(* CoDeSys 2.3.9.42 project: dev2.pro *)
(* Author: JvL *)
(* Libraries: ifm_RAWCan\ifm_RAWCan_NT_V020004.lib 7.6.24 16:48:07, ifm_CR0403\ifm_CR0403_V030400.lib 31.5.24 17:04:27, ifm_CANopen\ifm_NetVarLib_NT_V020004.lib 7.6.24 16:46:42, standard.lib 4.10.05 11:14:46, SysLibCallback.lib 7.6.24 16:43:25, 3S_CANOPENNETVAR.LIB 7.6.24 16:46:41, Iecsfc.lib 13.4.06 15:51:28, Util.lib 7.6.24 16:43:26, ifm_CANopen\3S_CANopenManager.lib 7.6.24 16:46:41, ifm_CANopen\3S_CanDrv.lib 7.6.24 16:46:41 *)

(* PLC configuration (modules and I/O channels)
Configuration [LocalConfiguration] node 0, in %IB0 out %QB0 {IFM_PARAM_WORD_TIME = 0}
AT %IB0 [ChInputBool] Input 00 Bit
AT %IB1 [ChInputBool] Input 01 Bit
AT %IB2 [ChInputBool] Input 02 Bit
AT %IB3 [ChInputBool] Input 03 Bit
IGNITION_KEY AT %IB4 [ChInputBool] Input 04 Bit
CHARGER_INPUT AT %IB5 [ChInputBool] Input 05 Bit
BATTERY1_IGNITION AT %IB6 [ChInputBool] Input 06 Bit
BATTERY2_IGNITION AT %IB7 [ChInputBool] Input 07 Bit
ARM_SWITCH AT %IB8 [ChInputBool] Input 08 Bit
KILL_SWITCH AT %IB9 [ChInputBool] Input 09 Bit
HYDRAULIC_SWITCH AT %IB10 [ChInputBool] Input 10 Bit
EM_SWITCH AT %IB11 [ChInputBool] Input 11 Bit
ARM_LED AT %QB0 [ChOutputBool] Output 00 Bit
PRECHARGE_RELAY AT %QB1 [ChOutputBool] Output 01 Bit
AT %QB2 [ChOutputBool] Output 02 Bit
BRAKE_LIGHT AT %QB3 [ChOutputBool] Output 03 Bit
EM_BRAKE AT %QB4 [ChOutputBool] Output 04 Bit
MCU_IGNITION AT %QB5 [ChOutputBool] Output 05 Bit
BATTERY1_RELAY AT %QB6 [ChOutputBool] Output 06 Bit
BATTERY2_RELAY AT %QB7 [ChOutputBool] Output 07 Bit
HORN AT %QB8 [ChOutputBool] Output 08 Bit
BUZZER AT %QB9 [ChOutputBool] Output 09 Bit
CONTACTOR AT %QB10 [ChOutputBool] Output 10 Bit
CHARGING_LED AT %QB11 [ChOutputBool] Output 11 Bit
System Inputs [LocalSystemInputs] node 2, in %IB12 out %QB12
  SUPPLY_VOLTAGE_VBBS AT %IW6 [ChInputWord] Supply voltage VBBS
  SUPPLY_VOLTAGE_VU AT %IW7 [ChInputWord] Supply voltage VU
  SUPPLY_VOLTAGE_VBB1 AT %IW8 [ChInputWord] Supply voltage VBB1
  SUPPLY_VOLTAGE_VBB2 AT %IW9 [ChInputWord] Supply voltage VBB2
  TEMPERATURE AT %IW10 [ChInputInt] Temperature
J1939 Interface [CAN_J1939] node 1, in %IB37 out %QB12
Interface CAN 2 [CAN_BUS] node 1, in %IB37 out %QB12 {STACK_DWORD_S = 0}
  J1939 Interface [CAN_J1939] node 1, in %IB37 out %QB12
*)

(* Global variable list: CanOpen implicit Variables *)
VAR_GLOBAL CONSTANT
	MAX_CTRLINDEX : INT := 0;
END_VAR

(* Global variable list: Global_Variables *)
VAR_GLOBAL
(*BATTERY*)
	BATTERY1_SOC: BYTE;
	BATTERY1_SOH: BYTE;
	BATTERY1_CHARGING: BOOL;
	BATTERY1_POWER: INT;
	BATTERY1_NTC1: BYTE;
	BATTERY1_NTC2: BYTE;
	BATTERY1_CAN_ERROR: BOOL;
	BATTERY1_CAPACITY: INT;
	BATTERY1_TOTAL_CAPACITY: INT;
	BATTERY1_CURRENT: INT;
	BATTERY1_FULLCHARGE_MIN: REAL;

	BATTERY2_SOC: BYTE;
	BATTERY2_SOH: BYTE;
	BATTERY2_CHARGING: BOOL;
	BATTERY2_POWER: INT;
	BATTERY2_NTC1: BYTE;
	BATTERY2_NTC2: BYTE;
	BATTERY2_CAN_ERROR: BOOL;
	BATTERY2_CAPACITY: INT;
	BATTERY2_TOTAL_CAPACITY: INT;
	BATTERY2_CURRENT: INT;
	BATTERY2_FULLCHARGE_MIN: REAL;

(*MCU <> MOTOR*)
	MOTOR_TARGET_RPM: ARRAY [1..6] OF INT;
	MOTOR_IGNITION: ARRAY [1..6] OF BOOL;

	MOTOR_RPM: ARRAY [1..6] OF INT;
	MOTOR_POWER: ARRAY [1..6] OF INT;
	MOTOR_PHASE_CURRENT: ARRAY [1..6] OF WORD;
	MOTOR_TEMPERATURE:ARRAY [1..6] OF BYTE;
	MCU_TEMPERATURE:ARRAY [1..6] OF BYTE;
	MCU_CAN_ERROR: ARRAY [1..6] OF BOOL;

	MOTOR1_FAULT_ARRAY: ARRAY [1..4] OF BYTE;
	MOTOR2_FAULT_ARRAY: ARRAY [1..4] OF BYTE;
	MOTOR6_FAULT_ARRAY: ARRAY [1..4] OF BYTE;
       MOTOR_OBD_ARRAY: ARRAY [1..6] OF WORD;

(*JOYSTICK*)
	LOG_JX: BYTE;
	LOG_JY: BYTE;
	JOY_ERROR: BOOL;
(*IMU*)
	X_ANGLE_BYTE:BYTE;
	Y_ANGLE_BYTE:BYTE;
	NEG_Y: BOOL;
	NEG_X: BOOL;
	Y_MAX_PEAK: BYTE;
	X_MAX_PEAK: BYTE;
	Y_MIN_PEAK: BYTE;
	X_MIN_PEAK: BYTE;
	IMU_CAN_ERROR:BOOL;
	IMU_ALERT: BOOL;
(*DISPLAY TELEMATICS*)
	HIGH_SPEED: BOOL;
	POWER_MODE: BOOL;
	HILL_HOLD: BOOL;
	DISABLE_MCU_CAN: BOOL;
	TRIP_RESET: BOOL;
      	BATTERY_CHARGING:BOOL;
(*MISC*)
	REVERSE: BOOL;
	MCU_BRAKE: BOOL;
(*HYDRAULICS*)
	HYDRAULIC_IGNITION: BOOL;
(*CALCULATIONS*)
	AVG_RPM: INT;
	RANGE_IN_KM: BYTE;
	SPEED: BYTE;

	RUNTIME: DWORD;
	HYDL_UP_TIME:DWORD;
	VEHICLE_UP_TIME: DWORD;
	VEHICLE_UP_TIME_LT: DWORD;

	ODO_KM: WORD;
	ODO_METER: DWORD;

	TRIP_METER: DWORD;
	TRIP_KM: WORD;

	DUMMY: BOOL;
END_VAR
VAR_GLOBAL RETAIN
	Y_MAX_RETAIN: BYTE;
	X_MAX_RETAIN: BYTE;
	Y_MIN_RETAIN: BYTE;
	X_MIN_RETAIN: BYTE;
END_VAR

(* Global variable list: Networkmanagement implicit Variables CAN *)
VAR_GLOBAL CONSTANT
	USE_NWVARS_CAN : BOOL := FALSE;
	MAX_NetVarItems_CAN	: INT := 0;
	MAX_NetVarPDO_Rx_CAN	: INT := 0;
	MAX_NetVarPDO_Tx_CAN	: INT := 0;
	MAX_NetVarOD_CAN		: INT := 0;
END_VAR
VAR_GLOBAL
	pNetVarItems_CAN		: ARRAY[0..MAX_NetVarItems_CAN] OF NetVarDataItem_CAN;
	pNetVarPDO_Rx_CAN		: ARRAY[0..MAX_NetVarPDO_Rx_CAN] OF NetVarPDO_Rx_CAN;
	pNetVarPDO_Tx_CAN		: ARRAY[0..MAX_NetVarPDO_Tx_CAN] OF NetVarPDO_Tx_CAN;
	pNetVarOD_CAN			: ARRAY[0..MAX_NetVarOD_CAN] OF NetVarOD_CAN;
END_VAR

(* POU PLC_PRG, FBD *)
PROGRAM PLC_PRG
VAR
	CONTACTOR_DELAY: TON;
END_VAR
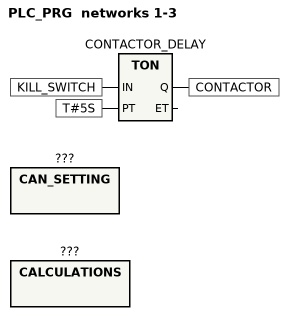
_FBD_ (* Function Block Diagram *)
NETWORK 1
	CONTACTOR_DELAY:TON(IN: KILL_SWITCH, PT: T#5S) => CONTACTOR
NETWORK 2
	???:CAN_SETTING()
NETWORK 3
	???:CALCULATIONS()
_END_FBD_
(* the same logic as Structured Text *)
(* Network 1 *)
CONTACTOR_DELAY(IN := KILL_SWITCH, PT := T#5S);
CONTACTOR := CONTACTOR_DELAY.Q;
(* Network 2: see the listing above *)
(* Network 3: see the listing above *)
END_PROGRAM

(* POU CAN_SETTING/CAN_SETTING, FBD *)
PROGRAM CAN_SETTING
(*
Created By: BHAGYESH
Date: 20-01-2024
Version: 1
Description: This program enables the CAN channels and sets the basic CAN parameter for both channels.
This block also controls the IFM's Inbuilt LED.
*)
VAR
	CAN_EN_1: CAN_ENABLE;
	CAN_EN_2: CAN_ENABLE;
	CAN_SET_1: CAN_SETDOWNLOADID;
	CAN_SET_2: CAN_SETDOWNLOADID;
	LED_SET: SET_LED;
	CAN_STATUS_1: CAN_STATUS;
	CAN_STATUS_2: CAN_STATUS;
	RESET_1: BOOL;
	RESET_2: BOOL;
END_VAR
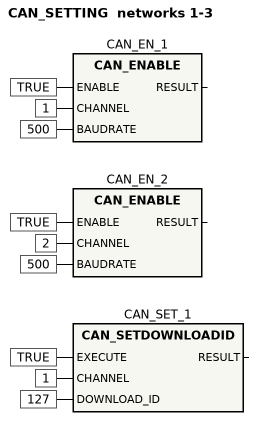
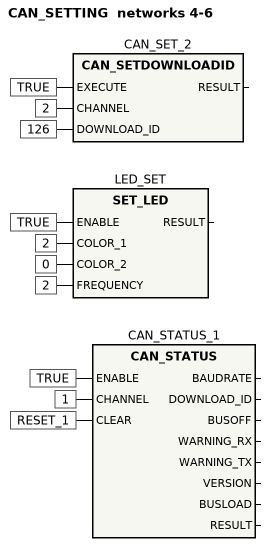
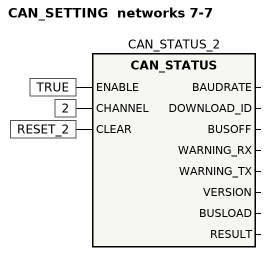
_FBD_ (* Function Block Diagram *)
NETWORK 1
	CAN_EN_1:CAN_ENABLE(ENABLE: TRUE, CHANNEL: 1, BAUDRATE: 500)
NETWORK 2
	CAN_EN_2:CAN_ENABLE(ENABLE: TRUE, CHANNEL: 2, BAUDRATE: 500)
NETWORK 3
	CAN_SET_1:CAN_SETDOWNLOADID(EXECUTE: TRUE, CHANNEL: 1, DOWNLOAD_ID: 127)
NETWORK 4
	CAN_SET_2:CAN_SETDOWNLOADID(EXECUTE: TRUE, CHANNEL: 2, DOWNLOAD_ID: 126)
NETWORK 5
	LED_SET:SET_LED(ENABLE: TRUE, COLOR_1: 2, COLOR_2: 0, FREQUENCY: 2)
NETWORK 6
	CAN_STATUS_1:CAN_STATUS(ENABLE: TRUE, CHANNEL: 1, CLEAR: RESET_1)
NETWORK 7
	CAN_STATUS_2:CAN_STATUS(ENABLE: TRUE, CHANNEL: 2, CLEAR: RESET_2)
_END_FBD_
(* the same logic as Structured Text *)
(* Network 1 *)
CAN_EN_1(ENABLE := TRUE, CHANNEL := 1, BAUDRATE := 500);
(* Network 2 *)
CAN_EN_2(ENABLE := TRUE, CHANNEL := 2, BAUDRATE := 500);
(* Network 3 *)
CAN_SET_1(EXECUTE := TRUE, CHANNEL := 1, DOWNLOAD_ID := 127);
(* Network 4 *)
CAN_SET_2(EXECUTE := TRUE, CHANNEL := 2, DOWNLOAD_ID := 126);
(* Network 5 *)
LED_SET(ENABLE := TRUE, COLOR_1 := 2, COLOR_2 := 0, FREQUENCY := 2);
(* Network 6 *)
CAN_STATUS_1(ENABLE := TRUE, CHANNEL := 1, CLEAR := RESET_1);
(* Network 7 *)
CAN_STATUS_2(ENABLE := TRUE, CHANNEL := 2, CLEAR := RESET_2);
END_PROGRAM

(* POU CALCULATIONS, LD *)
PROGRAM CALCULATIONS
VAR
(*SPEED*)
	ABS_RPM1: INT;
	ABS_RPM2: INT;
	RPM_SUM: INT;
	AVG_RPM_REAL: REAL;
	SPEED_REAL: REAL;

(* RUNTIME*)
	MOTOR_1_RUNNING: BOOL;
	MOTOR_2_RUNNING: BOOL;
	HYDRAULIC_HOURS: BOOL;
	COUNT_HOURS: BOOL;
	RISE: R_TRIG;
	FALL: F_TRIG;

	PREVIOUS_TIME: REAL;
	HYDL_PREVIOUS_TIME: REAL;
	VEHICLE_PREVIOUS_TIME: REAL;
	VEHICLE_PREVIOUS_TIME_LT: REAL;

	TON_RUNTIME: TON;
	ET_REAL: REAL;
	HOURS_RUN: REAL;

(*ODO & TRIP*)
	INSTANTANEOUS_DISTANCE: REAL;
	TIMER_ODO: TON;
	ODO_KM_DWORD: DWORD;

(*RANGE*)
	ACTUAL_CAPACITY: REAL;
	ODO_TARGET: DWORD;
	ODO_CYCLE_COMPLETE: BOOL;
	OLD_CAPACITY: REAL;
	DIFFERENCE: REAL;
	CAPACITY_FACTOR: REAL;
	TIMER_RISING: TP;

	HOLD_PREVIOUS_VALUE: BOOL;
	INITIAL_RANGE_REAL: REAL;
	REMAINING_CAPACITY: INT;
	BATTERY1_REMAINING_CAPACITY: INT;
	BATTERY1_FULLCHARGE_HOURS: REAL;
	BATTERY2_REMAINING_CAPACITY: INT;
	BATTERY2_FULLCHARGE_HOURS: REAL;
	TON_HYDL_RUNTIME: TON;
	HYDL_HOURS_RUN: REAL;
	ET_REAL_HYDL: REAL;
	RISE_2: R_TRIG;
	FAL0_2L: F_TRIG;
	FALL_2: F_TRIG;
	ABS_RPM6: INT;
	MINUTE_RUN: REAL;
	ODO_TRIP: DWORD;
	ODO_TRIP_METER: DWORD;
	TRIP_KM_REAL: REAL;
	TRIP_DWORD_KM: DWORD;
	VEHICLE_UP_TIME_COUNT: BOOL;
	RISE_3: R_TRIG;
	FALL_3: F_TRIG;
	TON_VEHICLE_RUNTIME: TON;
	ET_REAL_VEHICLE: REAL;
	VEHICLE_HOURS_RUN: REAL;
	RISE_4: R_TRIG;
	FALL_4: F_TRIG;
	VEHICLE_UP_TIME_COUNT_BW: BOOL;
	VEHICLE_UP_TIME_COUNT_LT: BOOL;
	TON_VEHICLE_RUNTIME_LT: TON;
	ET_REAL_VEHICLE_LT: REAL;
	VEHICLE_HOURS_RUN_LT: REAL;
END_VAR
VAR CONSTANT
	METER_CYCLE: DWORD := 500;						(*CHANGES BASED ON THE CALCULATION OF DISTANCE FACTOR*)
	SPEED_FACTOR: REAL:= 0.00146726;
	ODO_DISTANCE_FACTOR: REAL:= 0.0002037860;	(*GLX with 72.02 Gear Ratio - 500ms Cycle time*)
	ODO_TIME: TIME := T#485MS;							(*Actual calculation factor is for 500ms*)
END_VAR
VAR RETAIN
	RETAIN_DISTANCE: REAL:=457860;							(*In meter*)(*28_03_25 *)
	RETAIN_TIME: REAL := 800640000;			(*222.4 hour- 28-03-25*)	(*Final: REAL:= 3600000 ; //1hour  = 3600000*)
	HYDL_RETAIN_TIME: REAL:=414640000;             (*114.9 HR*)
	VEHICLE_RETAIN_TIME: REAL:=2160000;
	VEHICLE_RETAIN_TIME_LT: REAL:= 801720000;  (*222.7*)
	SUBTRACT_TRIP: DWORD;

END_VAR
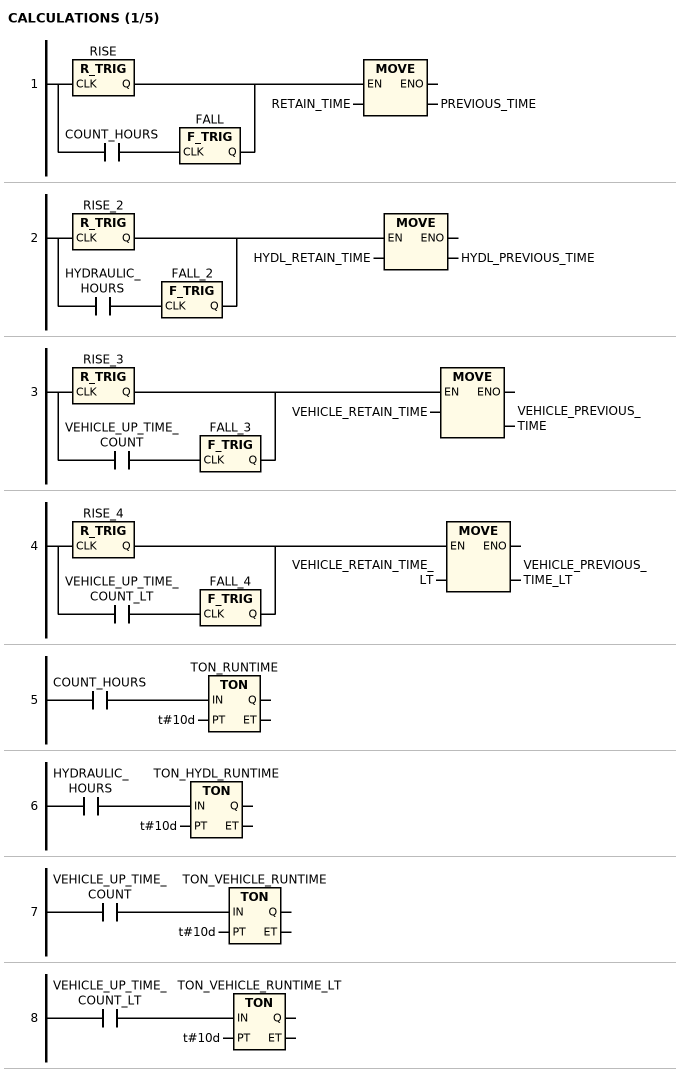
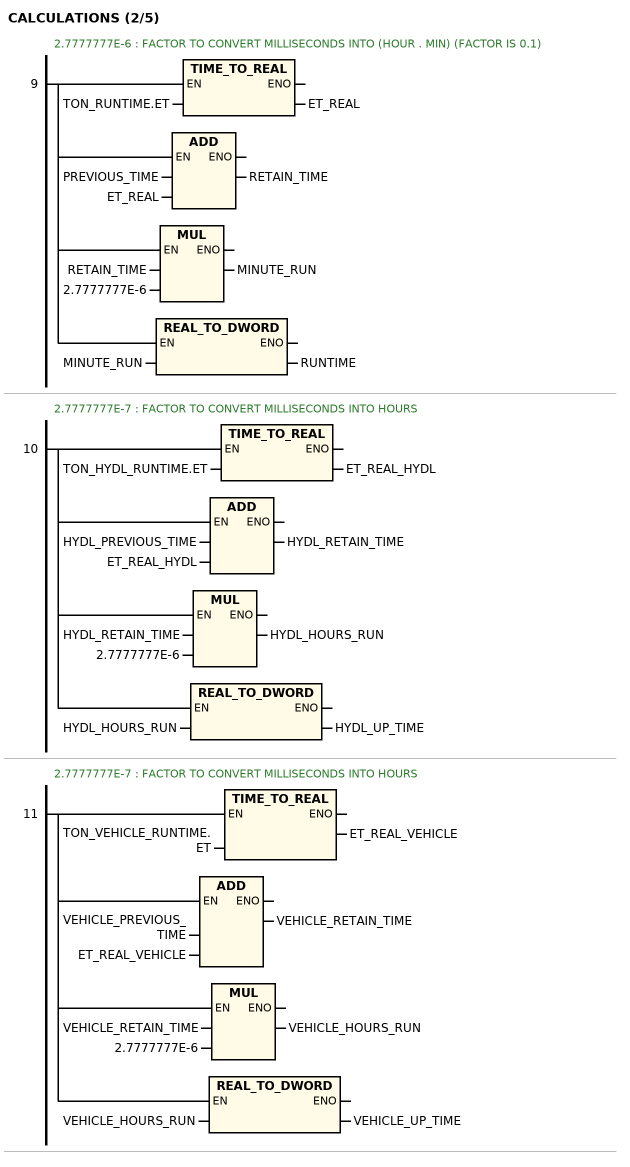
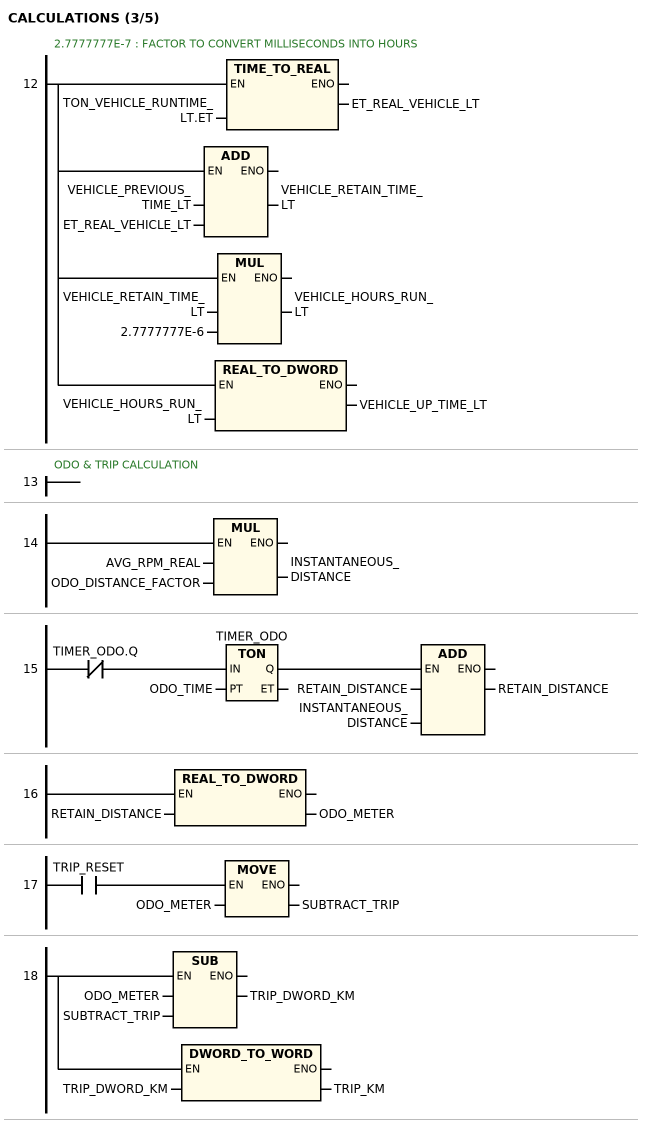
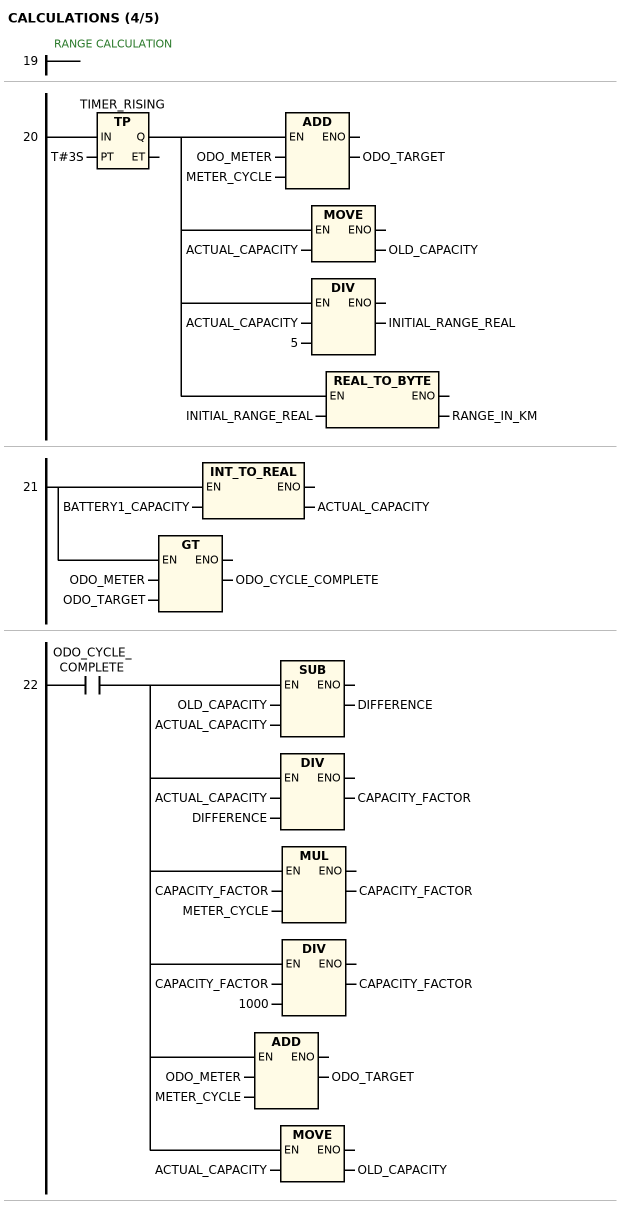
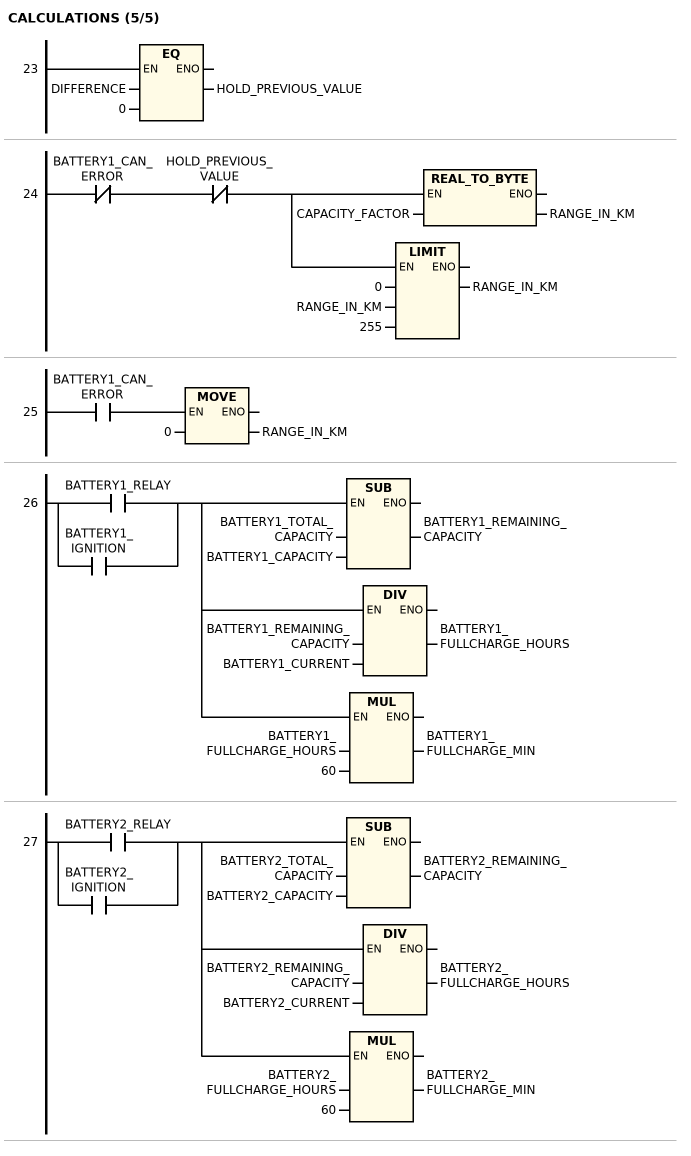
_LD_ (* Ladder Diagram *)
NETWORK 1
	{ RISE:R_TRIG(CLK: *) | [COUNT_HOURS] - FALL:F_TRIG(CLK: *) }
		EN --- MOVE(RETAIN_TIME) => PREVIOUS_TIME
NETWORK 2
	{ RISE_2:R_TRIG(CLK: *) | [HYDRAULIC_HOURS] - FALL_2:F_TRIG(CLK: *) }
		EN --- MOVE(HYDL_RETAIN_TIME) => HYDL_PREVIOUS_TIME
NETWORK 3
	{ RISE_3:R_TRIG(CLK: *) | [VEHICLE_UP_TIME_COUNT] - FALL_3:F_TRIG(CLK: *) }
		EN --- MOVE(VEHICLE_RETAIN_TIME) => VEHICLE_PREVIOUS_TIME
NETWORK 4
	{ RISE_4:R_TRIG(CLK: *) | [VEHICLE_UP_TIME_COUNT_LT] - FALL_4:F_TRIG(CLK: *) }
		EN --- MOVE(VEHICLE_RETAIN_TIME_LT) => VEHICLE_PREVIOUS_TIME_LT
NETWORK 5
	[COUNT_HOURS] - TON_RUNTIME:TON(IN: *, PT: t#10d)
NETWORK 6
	[HYDRAULIC_HOURS] - TON_HYDL_RUNTIME:TON(IN: *, PT: t#10d)
NETWORK 7
	[VEHICLE_UP_TIME_COUNT] - TON_VEHICLE_RUNTIME:TON(IN: *, PT: t#10d)
NETWORK 8
	[VEHICLE_UP_TIME_COUNT_LT] - TON_VEHICLE_RUNTIME_LT:TON(IN: *, PT: t#10d)
NETWORK 9 (* 2.7777777E-6 : FACTOR TO CONVERT MILLISECONDS INTO (HOUR . MIN) (FACTOR IS 0.1) *)
	*
		EN --- TIME_TO_REAL(TON_RUNTIME.ET) => ET_REAL
		EN --- ADD(PREVIOUS_TIME, ET_REAL) => RETAIN_TIME
		EN --- MUL(RETAIN_TIME, 2.7777777E-6) => MINUTE_RUN
		EN --- REAL_TO_DWORD(MINUTE_RUN) => RUNTIME
NETWORK 10 (* 2.7777777E-7 : FACTOR TO CONVERT MILLISECONDS INTO HOURS *)
	*
		EN --- TIME_TO_REAL(TON_HYDL_RUNTIME.ET) => ET_REAL_HYDL
		EN --- ADD(HYDL_PREVIOUS_TIME, ET_REAL_HYDL) => HYDL_RETAIN_TIME
		EN --- MUL(HYDL_RETAIN_TIME, 2.7777777E-6) => HYDL_HOURS_RUN
		EN --- REAL_TO_DWORD(HYDL_HOURS_RUN) => HYDL_UP_TIME
NETWORK 11 (* 2.7777777E-7 : FACTOR TO CONVERT MILLISECONDS INTO HOURS *)
	*
		EN --- TIME_TO_REAL(TON_VEHICLE_RUNTIME.ET) => ET_REAL_VEHICLE
		EN --- ADD(VEHICLE_PREVIOUS_TIME, ET_REAL_VEHICLE) => VEHICLE_RETAIN_TIME
		EN --- MUL(VEHICLE_RETAIN_TIME, 2.7777777E-6) => VEHICLE_HOURS_RUN
		EN --- REAL_TO_DWORD(VEHICLE_HOURS_RUN) => VEHICLE_UP_TIME
NETWORK 12 (* 2.7777777E-7 : FACTOR TO CONVERT MILLISECONDS INTO HOURS *)
	*
		EN --- TIME_TO_REAL(TON_VEHICLE_RUNTIME_LT.ET) => ET_REAL_VEHICLE_LT
		EN --- ADD(VEHICLE_PREVIOUS_TIME_LT, ET_REAL_VEHICLE_LT) => VEHICLE_RETAIN_TIME_LT
		EN --- MUL(VEHICLE_RETAIN_TIME_LT, 2.7777777E-6) => VEHICLE_HOURS_RUN_LT
		EN --- REAL_TO_DWORD(VEHICLE_HOURS_RUN_LT) => VEHICLE_UP_TIME_LT
NETWORK 13 (* ODO & TRIP CALCULATION *)
	*
NETWORK 14
	*
		EN --- MUL(AVG_RPM_REAL, ODO_DISTANCE_FACTOR) => INSTANTANEOUS_DISTANCE
NETWORK 15
	[/TIMER_ODO.Q] - TIMER_ODO:TON(IN: *, PT: ODO_TIME)
		EN --- ADD(RETAIN_DISTANCE, INSTANTANEOUS_DISTANCE) => RETAIN_DISTANCE
NETWORK 16
	*
		EN --- REAL_TO_DWORD(RETAIN_DISTANCE) => ODO_METER
NETWORK 17
	[TRIP_RESET]
		EN --- MOVE(ODO_METER) => SUBTRACT_TRIP
NETWORK 18
	*
		EN --- SUB(ODO_METER, SUBTRACT_TRIP) => TRIP_DWORD_KM
		EN --- DWORD_TO_WORD(TRIP_DWORD_KM) => TRIP_KM
NETWORK 19 (* RANGE CALCULATION *)
	*
NETWORK 20
	TIMER_RISING:TP(IN: *, PT: T#3S)
		EN --- ADD(ODO_METER, METER_CYCLE) => ODO_TARGET
		EN --- MOVE(ACTUAL_CAPACITY) => OLD_CAPACITY
		EN --- DIV(ACTUAL_CAPACITY, 5) => INITIAL_RANGE_REAL
		EN --- REAL_TO_BYTE(INITIAL_RANGE_REAL) => RANGE_IN_KM
NETWORK 21
	*
		EN --- INT_TO_REAL(BATTERY1_CAPACITY) => ACTUAL_CAPACITY
		EN --- GT(ODO_METER, ODO_TARGET) => ODO_CYCLE_COMPLETE
NETWORK 22
	[ODO_CYCLE_COMPLETE]
		EN --- SUB(OLD_CAPACITY, ACTUAL_CAPACITY) => DIFFERENCE
		EN --- DIV(ACTUAL_CAPACITY, DIFFERENCE) => CAPACITY_FACTOR
		EN --- MUL(CAPACITY_FACTOR, METER_CYCLE) => CAPACITY_FACTOR
		EN --- DIV(CAPACITY_FACTOR, 1000) => CAPACITY_FACTOR
		EN --- ADD(ODO_METER, METER_CYCLE) => ODO_TARGET
		EN --- MOVE(ACTUAL_CAPACITY) => OLD_CAPACITY
NETWORK 23
	*
		EN --- EQ(DIFFERENCE, 0) => HOLD_PREVIOUS_VALUE
NETWORK 24
	[/BATTERY1_CAN_ERROR] - [/HOLD_PREVIOUS_VALUE]
		EN --- REAL_TO_BYTE(CAPACITY_FACTOR) => RANGE_IN_KM
		EN --- LIMIT(0, RANGE_IN_KM, 255) => RANGE_IN_KM
NETWORK 25
	[BATTERY1_CAN_ERROR]
		EN --- MOVE(0) => RANGE_IN_KM
NETWORK 26
	{ [BATTERY1_RELAY] | [BATTERY1_IGNITION] }
		EN --- SUB(BATTERY1_TOTAL_CAPACITY, BATTERY1_CAPACITY) => BATTERY1_REMAINING_CAPACITY
		EN --- DIV(BATTERY1_REMAINING_CAPACITY, BATTERY1_CURRENT) => BATTERY1_FULLCHARGE_HOURS
		EN --- MUL(BATTERY1_FULLCHARGE_HOURS, 60) => BATTERY1_FULLCHARGE_MIN
NETWORK 27
	{ [BATTERY2_RELAY] | [BATTERY2_IGNITION] }
		EN --- SUB(BATTERY2_TOTAL_CAPACITY, BATTERY2_CAPACITY) => BATTERY2_REMAINING_CAPACITY
		EN --- DIV(BATTERY2_REMAINING_CAPACITY, BATTERY2_CURRENT) => BATTERY2_FULLCHARGE_HOURS
		EN --- MUL(BATTERY2_FULLCHARGE_HOURS, 60) => BATTERY2_FULLCHARGE_MIN
_END_LD_
(* the same logic as Structured Text *)
(* Network 1 *)
RISE(CLK := TRUE);
FALL(CLK := COUNT_HOURS);
IF RISE.Q OR FALL.Q THEN
	PREVIOUS_TIME := RETAIN_TIME;
END_IF;
(* Network 2 *)
RISE_2(CLK := TRUE);
FALL_2(CLK := HYDRAULIC_HOURS);
IF RISE_2.Q OR FALL_2.Q THEN
	HYDL_PREVIOUS_TIME := HYDL_RETAIN_TIME;
END_IF;
(* Network 3 *)
RISE_3(CLK := TRUE);
FALL_3(CLK := VEHICLE_UP_TIME_COUNT);
IF RISE_3.Q OR FALL_3.Q THEN
	VEHICLE_PREVIOUS_TIME := VEHICLE_RETAIN_TIME;
END_IF;
(* Network 4 *)
RISE_4(CLK := TRUE);
FALL_4(CLK := VEHICLE_UP_TIME_COUNT_LT);
IF RISE_4.Q OR FALL_4.Q THEN
	VEHICLE_PREVIOUS_TIME_LT := VEHICLE_RETAIN_TIME_LT;
END_IF;
(* Network 5 *)
TON_RUNTIME(IN := COUNT_HOURS, PT := t#10d);
(* Network 6 *)
TON_HYDL_RUNTIME(IN := HYDRAULIC_HOURS, PT := t#10d);
(* Network 7 *)
TON_VEHICLE_RUNTIME(IN := VEHICLE_UP_TIME_COUNT, PT := t#10d);
(* Network 8 *)
TON_VEHICLE_RUNTIME_LT(IN := VEHICLE_UP_TIME_COUNT_LT, PT := t#10d);
(* Network 9: 2.7777777E-6 : FACTOR TO CONVERT MILLISECONDS INTO (HOUR . MIN) (FACTOR IS 0.1) *)
ET_REAL := TIME_TO_REAL(TON_RUNTIME.ET);
RETAIN_TIME := PREVIOUS_TIME + ET_REAL;
MINUTE_RUN := RETAIN_TIME * (2.7777777E-6);
RUNTIME := REAL_TO_DWORD(MINUTE_RUN);
(* Network 10: 2.7777777E-7 : FACTOR TO CONVERT MILLISECONDS INTO HOURS *)
ET_REAL_HYDL := TIME_TO_REAL(TON_HYDL_RUNTIME.ET);
HYDL_RETAIN_TIME := HYDL_PREVIOUS_TIME + ET_REAL_HYDL;
HYDL_HOURS_RUN := HYDL_RETAIN_TIME * (2.7777777E-6);
HYDL_UP_TIME := REAL_TO_DWORD(HYDL_HOURS_RUN);
(* Network 11: 2.7777777E-7 : FACTOR TO CONVERT MILLISECONDS INTO HOURS *)
ET_REAL_VEHICLE := TIME_TO_REAL(TON_VEHICLE_RUNTIME.ET);
VEHICLE_RETAIN_TIME := VEHICLE_PREVIOUS_TIME + ET_REAL_VEHICLE;
VEHICLE_HOURS_RUN := VEHICLE_RETAIN_TIME * (2.7777777E-6);
VEHICLE_UP_TIME := REAL_TO_DWORD(VEHICLE_HOURS_RUN);
(* Network 12: 2.7777777E-7 : FACTOR TO CONVERT MILLISECONDS INTO HOURS *)
ET_REAL_VEHICLE_LT := TIME_TO_REAL(TON_VEHICLE_RUNTIME_LT.ET);
VEHICLE_RETAIN_TIME_LT := VEHICLE_PREVIOUS_TIME_LT + ET_REAL_VEHICLE_LT;
VEHICLE_HOURS_RUN_LT := VEHICLE_RETAIN_TIME_LT * (2.7777777E-6);
VEHICLE_UP_TIME_LT := REAL_TO_DWORD(VEHICLE_HOURS_RUN_LT);
(* Network 13: ODO & TRIP CALCULATION *)
(* Network 14 *)
INSTANTANEOUS_DISTANCE := AVG_RPM_REAL * ODO_DISTANCE_FACTOR;
(* Network 15 *)
TIMER_ODO(IN := NOT TIMER_ODO.Q, PT := ODO_TIME);
IF TIMER_ODO.Q THEN
	RETAIN_DISTANCE := RETAIN_DISTANCE + INSTANTANEOUS_DISTANCE;
END_IF;
(* Network 16 *)
ODO_METER := REAL_TO_DWORD(RETAIN_DISTANCE);
(* Network 17 *)
IF TRIP_RESET THEN
	SUBTRACT_TRIP := ODO_METER;
END_IF;
(* Network 18 *)
TRIP_DWORD_KM := ODO_METER - SUBTRACT_TRIP;
TRIP_KM := DWORD_TO_WORD(TRIP_DWORD_KM);
(* Network 19: RANGE CALCULATION *)
(* Network 20 *)
TIMER_RISING(IN := TRUE, PT := T#3S);
IF TIMER_RISING.Q THEN
	ODO_TARGET := ODO_METER + METER_CYCLE;
	OLD_CAPACITY := ACTUAL_CAPACITY;
	INITIAL_RANGE_REAL := ACTUAL_CAPACITY / 5;
	RANGE_IN_KM := REAL_TO_BYTE(INITIAL_RANGE_REAL);
END_IF;
(* Network 21 *)
ACTUAL_CAPACITY := INT_TO_REAL(BATTERY1_CAPACITY);
ODO_CYCLE_COMPLETE := ODO_METER > ODO_TARGET;
(* Network 22 *)
IF ODO_CYCLE_COMPLETE THEN
	DIFFERENCE := OLD_CAPACITY - ACTUAL_CAPACITY;
	CAPACITY_FACTOR := ACTUAL_CAPACITY / DIFFERENCE;
	CAPACITY_FACTOR := CAPACITY_FACTOR * METER_CYCLE;
	CAPACITY_FACTOR := CAPACITY_FACTOR / 1000;
	ODO_TARGET := ODO_METER + METER_CYCLE;
	OLD_CAPACITY := ACTUAL_CAPACITY;
END_IF;
(* Network 23 *)
HOLD_PREVIOUS_VALUE := DIFFERENCE = 0;
(* Network 24 *)
IF NOT BATTERY1_CAN_ERROR AND NOT HOLD_PREVIOUS_VALUE THEN
	RANGE_IN_KM := REAL_TO_BYTE(CAPACITY_FACTOR);
	RANGE_IN_KM := LIMIT(0, RANGE_IN_KM, 255);
END_IF;
(* Network 25 *)
IF BATTERY1_CAN_ERROR THEN
	RANGE_IN_KM := 0;
END_IF;
(* Network 26 *)
IF BATTERY1_RELAY OR BATTERY1_IGNITION THEN
	BATTERY1_REMAINING_CAPACITY := BATTERY1_TOTAL_CAPACITY - BATTERY1_CAPACITY;
	BATTERY1_FULLCHARGE_HOURS := BATTERY1_REMAINING_CAPACITY / BATTERY1_CURRENT;
	BATTERY1_FULLCHARGE_MIN := BATTERY1_FULLCHARGE_HOURS * 60;
END_IF;
(* Network 27 *)
IF BATTERY2_RELAY OR BATTERY2_IGNITION THEN
	BATTERY2_REMAINING_CAPACITY := BATTERY2_TOTAL_CAPACITY - BATTERY2_CAPACITY;
	BATTERY2_FULLCHARGE_HOURS := BATTERY2_REMAINING_CAPACITY / BATTERY2_CURRENT;
	BATTERY2_FULLCHARGE_MIN := BATTERY2_FULLCHARGE_HOURS * 60;
END_IF;
END_PROGRAM

(* POU FB_LIBRARY/ALTERNATE, LD *)
FUNCTION_BLOCK ALTERNATE
VAR_INPUT
	IN: BOOL;
END_VAR
VAR_OUTPUT
	OUT: BOOL;
END_VAR
VAR
	S1: BOOL;
	S2: BOOL;
END_VAR
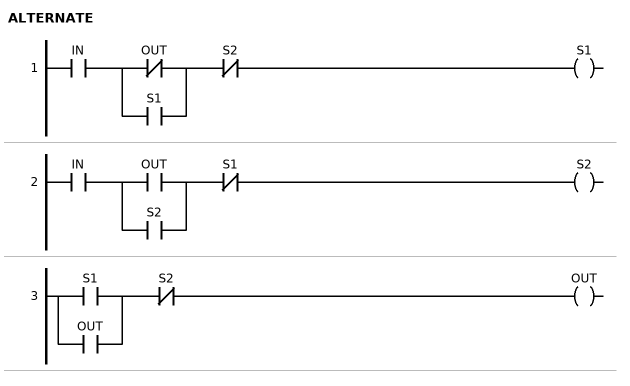
_LD_ (* Ladder Diagram *)
NETWORK 1
	[IN] - { [/OUT] | [S1] } - [/S2] --- (S1)
NETWORK 2
	[IN] - { [OUT] | [S2] } - [/S1] --- (S2)
NETWORK 3
	{ [S1] | [OUT] } - [/S2] --- (OUT)
_END_LD_
(* the same logic as Structured Text *)
(* Network 1 *)
S1 := IN AND (NOT OUT OR S1) AND NOT S2;
(* Network 2 *)
S2 := IN AND (OUT OR S2) AND NOT S1;
(* Network 3 *)
OUT := (S1 OR OUT) AND NOT S2;
END_FUNCTION_BLOCK

(* POU PROGRAM_FBs/ARM_LOGIC, LD *)
FUNCTION_BLOCK ARM_LOGIC
VAR_INPUT
	ARM_INPUT: BOOL;
	DISARM: BOOL;
	POST_IN: BOOL;
END_VAR
VAR_OUTPUT
	ARM: BOOL;
	ARMLED: BOOL;
END_VAR
VAR
	DELAY: TON;
	S1: BOOL;
	S2: BOOL;
	BLINKY: BLINK;
END_VAR
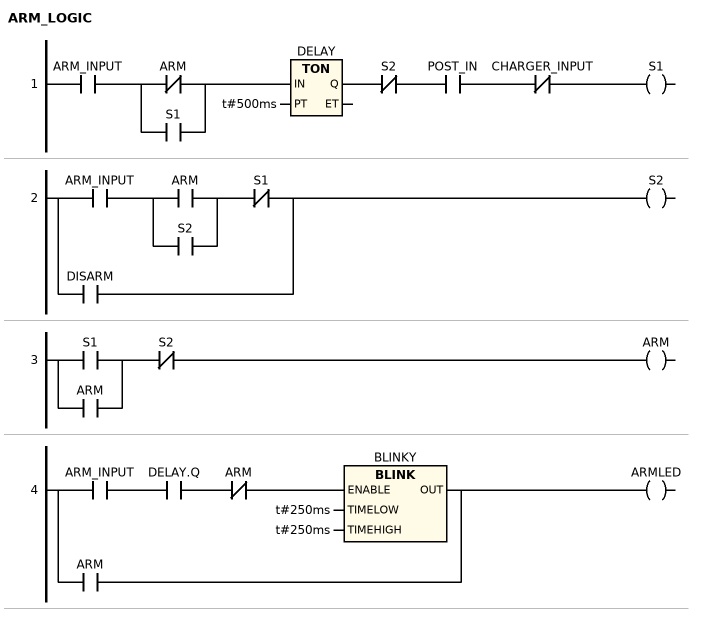
_LD_ (* Ladder Diagram *)
NETWORK 1
	[ARM_INPUT] - { [/ARM] | [S1] } - DELAY:TON(IN: *, PT: t#500ms) - [/S2] - [POST_IN] - [/CHARGER_INPUT] --- (S1)
NETWORK 2
	{ [ARM_INPUT] - { [ARM] | [S2] } - [/S1] | [DISARM] } --- (S2)
NETWORK 3
	{ [S1] | [ARM] } - [/S2] --- (ARM)
NETWORK 4
	{ [ARM_INPUT] - [DELAY.Q] - [/ARM] - BLINKY:BLINK(ENABLE: *, TIMELOW: t#250ms, TIMEHIGH: t#250ms) | [ARM] } --- (ARMLED)
_END_LD_
(* the same logic as Structured Text *)
(* Network 1 *)
DELAY(IN := ARM_INPUT AND (NOT ARM OR S1), PT := t#500ms);
S1 := DELAY.Q AND NOT S2 AND POST_IN AND NOT CHARGER_INPUT;
(* Network 2 *)
S2 := ARM_INPUT AND (ARM OR S2) AND NOT S1 OR DISARM;
(* Network 3 *)
ARM := (S1 OR ARM) AND NOT S2;
(* Network 4 *)
BLINKY(ENABLE := ARM_INPUT AND DELAY.Q AND NOT ARM, TIMELOW := t#250ms, TIMEHIGH := t#250ms);
ARMLED := BLINKY.OUT OR ARM;
END_FUNCTION_BLOCK

(* POU FUNCTIONS/BYTE_WORD_FUNCTION, ST *)
FUNCTION BYTE_WORD_FUNCTION : WORD
(*
Created by: Bhagyesh Unadkat
Date: 29-03-24
Version: 1
Updated by:
Update date:
Description: This block merges Two bytes of data into WORD data.
*)
VAR_INPUT
	BYTE_H: BYTE;
	BYTE_L: BYTE;
END_VAR
VAR
	MSB: WORD;
END_VAR
MSB:= BYTE_H * 256;
BYTE_WORD_FUNCTION:= MSB + BYTE_L;
END_FUNCTION

(* POU MCU/CHARA_MCU_RX, LD *)
FUNCTION_BLOCK CHARA_MCU_RX
(*
Created by: Bhagyesh Unadkat
Date: 11-09-24
Version: 5
Updated by: Karthik
Update date: 08-03-25
Description: This block receives CAN data from CHARA MCU.

		***Updates***
V2
	DC current and POWER added.
V3   
	Added OBD Code and adjusted the fault array accordingly.
	CAN error added to OBD code MSB bit as it is 12-bit value.
V4 
	Taken Motor Ignition as VAR_INPUT to reset RPM AND POWER TO 0
V5
	Converted CURRENT raw values from word to int, and then dividing by 1000.
V6
	Unmerged CAN error and OBD code.
V7
	Making OBD code zero when theres is a CAN error. 

FAULT ARRAY [DATATYPE: BYTE]
[1] MSG-2 BYTE2 and MSG-5 BYTE3		
		BYTE [BIT 0..7]: MSG2BYTE2 (BIT_0 TO BIT_2)------- AND-------- MSG5BYTE3 (BIT_0 TO BIT_4)
[2] MSG 2 :BYTE 7
[3] MSG 5: BYTE 2
[4] MSG 5: BYTE 4
*)
VAR_INPUT
	IGNITION: BOOL;
	MOTOR_IGNITION: BOOL;
	CAN_CHANNEL: BYTE;
	ID_1: DWORD;
	ID_2: DWORD;
	ID_4: DWORD;
	ID_5: DWORD;
	ID_6: DWORD;
END_VAR
VAR_OUTPUT
	RPM: INT;
	POWER: INT;
	PHASE_CURRENT: WORD;
	M_TEMP: BYTE;
	C_TEMP: BYTE;
	OBD_CODE: WORD;
	FAULT_ARRAY: ARRAY [1..4] OF BYTE;
	CAN_ERROR: BOOL;
END_VAR
VAR
	RX_1: RX_CAN;
	RX_2: RX_CAN;
	RX_4: RX_CAN;
	RX_5: RX_CAN;
	RX_6: RX_CAN;
	TIMER_ERROR: TON;

	RPM_WORD: WORD;
	PHASE_WORD: WORD;
	REVERSE_DIRECTION: BOOL;
	DIR_FACTOR: INT;
	DELAY: TON;
	RPM_INT: INT;
	CURRENT_WORD: WORD;
	CURRENT_INT: INT;
	VOLTAGE_INT: INT;
	RPM_SIGNED: INT;
	POWER_INT: INT;
END_VAR
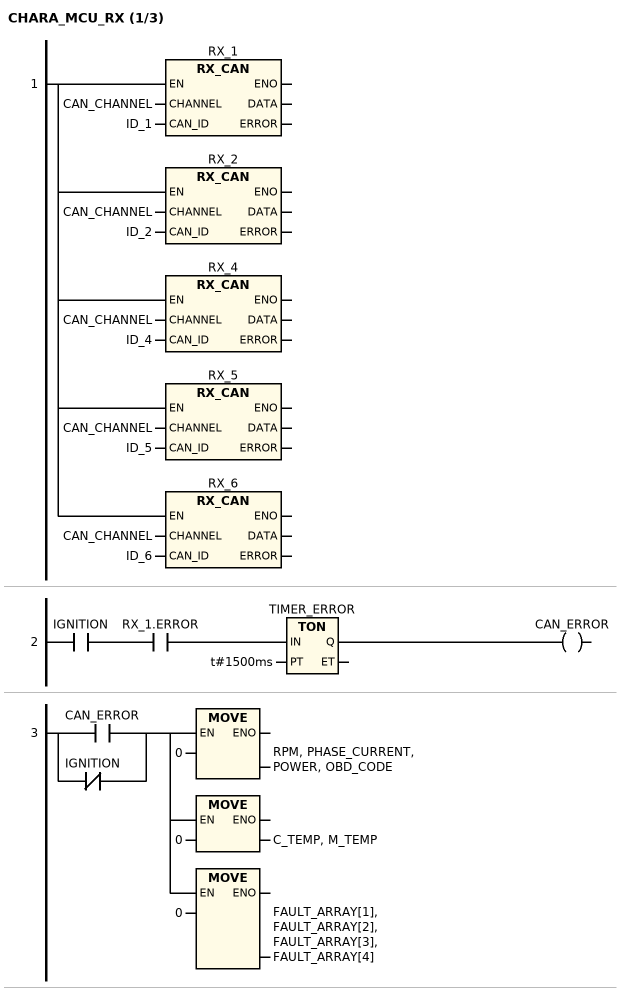
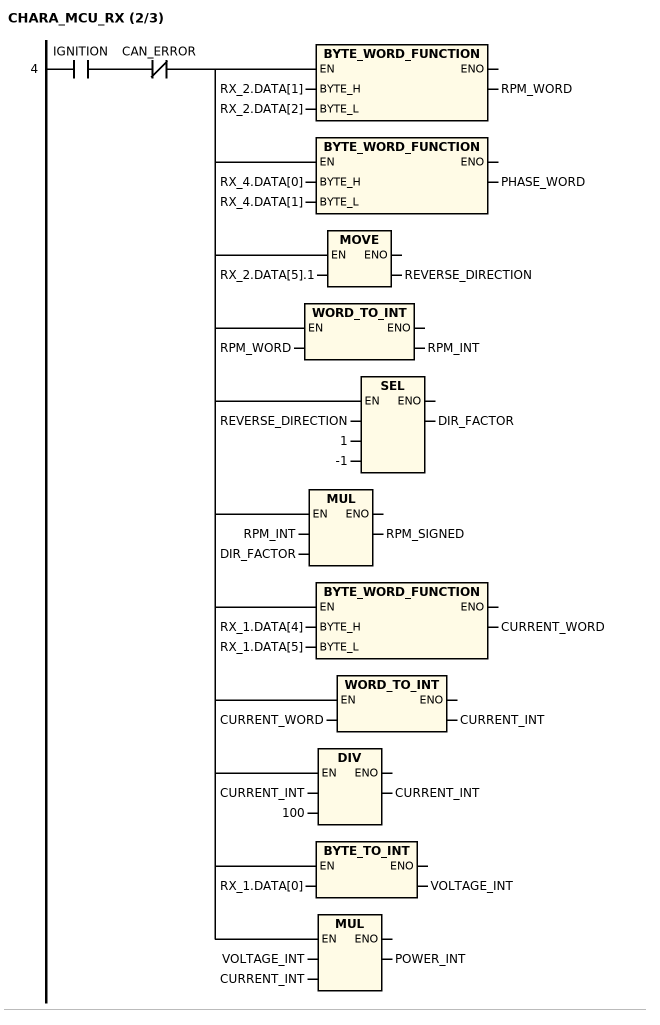
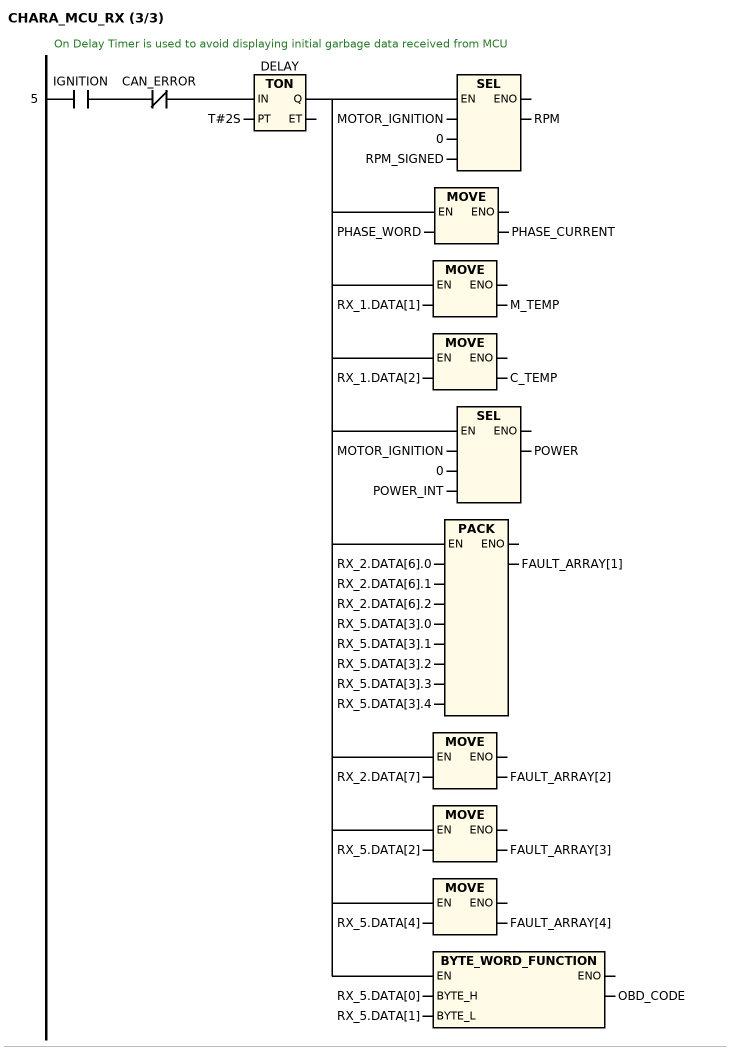
_LD_ (* Ladder Diagram *)
NETWORK 1
	*
		EN --- RX_1:RX_CAN(CHANNEL: CAN_CHANNEL, CAN_ID: ID_1)
		EN --- RX_2:RX_CAN(CHANNEL: CAN_CHANNEL, CAN_ID: ID_2)
		EN --- RX_4:RX_CAN(CHANNEL: CAN_CHANNEL, CAN_ID: ID_4)
		EN --- RX_5:RX_CAN(CHANNEL: CAN_CHANNEL, CAN_ID: ID_5)
		EN --- RX_6:RX_CAN(CHANNEL: CAN_CHANNEL, CAN_ID: ID_6)
NETWORK 2
	[IGNITION] - [RX_1.ERROR] - TIMER_ERROR:TON(IN: *, PT: t#1500ms) --- (CAN_ERROR)
NETWORK 3
	{ [CAN_ERROR] | [/IGNITION] }
		EN --- MOVE(0) => RPM, PHASE_CURRENT, POWER, OBD_CODE
		EN --- MOVE(0) => C_TEMP, M_TEMP
		EN --- MOVE(0) => FAULT_ARRAY[1], FAULT_ARRAY[2], FAULT_ARRAY[3], FAULT_ARRAY[4]
NETWORK 4
	[IGNITION] - [/CAN_ERROR]
		EN --- BYTE_WORD_FUNCTION(BYTE_H: RX_2.DATA[1], BYTE_L: RX_2.DATA[2]) => RPM_WORD
		EN --- BYTE_WORD_FUNCTION(BYTE_H: RX_4.DATA[0], BYTE_L: RX_4.DATA[1]) => PHASE_WORD
		EN --- MOVE(RX_2.DATA[5].1) => REVERSE_DIRECTION
		EN --- WORD_TO_INT(RPM_WORD) => RPM_INT
		EN --- SEL(REVERSE_DIRECTION, 1, -1) => DIR_FACTOR
		EN --- MUL(RPM_INT, DIR_FACTOR) => RPM_SIGNED
		EN --- BYTE_WORD_FUNCTION(BYTE_H: RX_1.DATA[4], BYTE_L: RX_1.DATA[5]) => CURRENT_WORD
		EN --- WORD_TO_INT(CURRENT_WORD) => CURRENT_INT
		EN --- DIV(CURRENT_INT, 100) => CURRENT_INT
		EN --- BYTE_TO_INT(RX_1.DATA[0]) => VOLTAGE_INT
		EN --- MUL(VOLTAGE_INT, CURRENT_INT) => POWER_INT
NETWORK 5 (* On Delay Timer is used to avoid displaying initial garbage data received from MCU *)
	[IGNITION] - [/CAN_ERROR] - DELAY:TON(IN: *, PT: T#2S)
		EN --- SEL(MOTOR_IGNITION, 0, RPM_SIGNED) => RPM
		EN --- MOVE(PHASE_WORD) => PHASE_CURRENT
		EN --- MOVE(RX_1.DATA[1]) => M_TEMP
		EN --- MOVE(RX_1.DATA[2]) => C_TEMP
		EN --- SEL(MOTOR_IGNITION, 0, POWER_INT) => POWER
		EN --- PACK(RX_2.DATA[6].0, RX_2.DATA[6].1, RX_2.DATA[6].2, RX_5.DATA[3].0, RX_5.DATA[3].1, RX_5.DATA[3].2, RX_5.DATA[3].3, RX_5.DATA[3].4) => FAULT_ARRAY[1]
		EN --- MOVE(RX_2.DATA[7]) => FAULT_ARRAY[2]
		EN --- MOVE(RX_5.DATA[2]) => FAULT_ARRAY[3]
		EN --- MOVE(RX_5.DATA[4]) => FAULT_ARRAY[4]
		EN --- BYTE_WORD_FUNCTION(BYTE_H: RX_5.DATA[0], BYTE_L: RX_5.DATA[1]) => OBD_CODE
_END_LD_
(* the same logic as Structured Text *)
(* Network 1 *)
RX_1(CHANNEL := CAN_CHANNEL, CAN_ID := ID_1);
RX_2(CHANNEL := CAN_CHANNEL, CAN_ID := ID_2);
RX_4(CHANNEL := CAN_CHANNEL, CAN_ID := ID_4);
RX_5(CHANNEL := CAN_CHANNEL, CAN_ID := ID_5);
RX_6(CHANNEL := CAN_CHANNEL, CAN_ID := ID_6);
(* Network 2 *)
TIMER_ERROR(IN := IGNITION AND RX_1.ERROR, PT := t#1500ms);
CAN_ERROR := TIMER_ERROR.Q;
(* Network 3: see the listing above *)
(* Network 4 *)
IF IGNITION AND NOT CAN_ERROR THEN
	RPM_WORD := BYTE_WORD_FUNCTION(BYTE_H := RX_2.DATA[1], BYTE_L := RX_2.DATA[2]);
	PHASE_WORD := BYTE_WORD_FUNCTION(BYTE_H := RX_4.DATA[0], BYTE_L := RX_4.DATA[1]);
	REVERSE_DIRECTION := RX_2.DATA[5].1;
	RPM_INT := WORD_TO_INT(RPM_WORD);
	DIR_FACTOR := SEL(REVERSE_DIRECTION, 1, -1);
	RPM_SIGNED := RPM_INT * DIR_FACTOR;
	CURRENT_WORD := BYTE_WORD_FUNCTION(BYTE_H := RX_1.DATA[4], BYTE_L := RX_1.DATA[5]);
	CURRENT_INT := WORD_TO_INT(CURRENT_WORD);
	CURRENT_INT := CURRENT_INT / 100;
	VOLTAGE_INT := BYTE_TO_INT(RX_1.DATA[0]);
	POWER_INT := VOLTAGE_INT * CURRENT_INT;
END_IF;
(* Network 5 *)
DELAY(IN := IGNITION AND NOT CAN_ERROR, PT := T#2S);
IF DELAY.Q THEN
	RPM := SEL(MOTOR_IGNITION, 0, RPM_SIGNED);
	PHASE_CURRENT := PHASE_WORD;
	M_TEMP := RX_1.DATA[1];
	C_TEMP := RX_1.DATA[2];
	POWER := SEL(MOTOR_IGNITION, 0, POWER_INT);
	FAULT_ARRAY[1] := PACK(RX_2.DATA[6].0, RX_2.DATA[6].1, RX_2.DATA[6].2, RX_5.DATA[3].0, RX_5.DATA[3].1, RX_5.DATA[3].2, RX_5.DATA[3].3, RX_5.DATA[3].4);
	FAULT_ARRAY[2] := RX_2.DATA[7];
	FAULT_ARRAY[3] := RX_5.DATA[2];
	FAULT_ARRAY[4] := RX_5.DATA[4];
	OBD_CODE := BYTE_WORD_FUNCTION(BYTE_H := RX_5.DATA[0], BYTE_L := RX_5.DATA[1]);
END_IF;
END_FUNCTION_BLOCK

(* POU FB_LIBRARY/RX_CAN, CFC *)
FUNCTION_BLOCK RX_CAN
(*
Created By: BHAGYESH
Date: 1-10-2023
Version: 1
Description: This function block checks the CAN data and updates the output CAN data only when it receives the new data.
*)
VAR_INPUT
	CHANNEL: BYTE;
	CAN_ID: DWORD;
END_VAR
VAR_OUTPUT
	DATA: ARRAY [0..7] OF BYTE;
	ERROR: BOOL;
END_VAR
VAR
	Rx: CAN_RX;

END_VAR
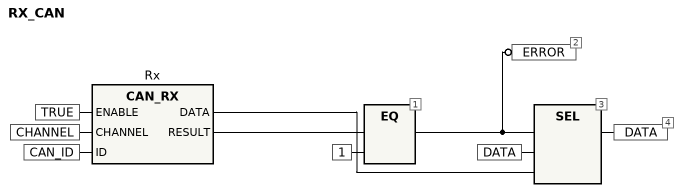
_CFC_ (* Continuous Function Chart, elements in execution order *)
#0 Rx:CAN_RX(ENABLE: TRUE, CHANNEL: CHANNEL, ID: CAN_ID)
#1 EQ(#0.RESULT, 1)
#2 ERROR <= NOT #1
#3 SEL(#1, DATA, #0.DATA)
#4 DATA <= #3
_END_CFC_
(* the same logic as Structured Text *)
Rx(ENABLE := TRUE, CHANNEL := CHANNEL, ID := CAN_ID);
ERROR := NOT (Rx.RESULT = 1);
DATA := SEL(Rx.RESULT = 1, DATA, Rx.DATA);
END_FUNCTION_BLOCK

(* POU MCU/CHARA_MCU_TX, LD *)
FUNCTION_BLOCK CHARA_MCU_TX
(*
Created by: Bhagyesh Unadkat
Date: Sep 11, 2024
Version: 4
Updated by: Bhagyesh
Update date: Dec 13, 2024
Description: This block transmits CAN data to the CHARA MCU to control the motor.

NOTE:  BIG ENDIAN FORMAT

Byte0 & Byte1: Signed RPM Big Endian format (-6000 to 6000)
Byte2: Ignition State =  0 & 1 (OFF and ON respectively)
Byte3: Phase Current Limit (%) = 0 - 100
Byte4: Regen (%) = 0 - 100 (Not configured yet)
Byte5: Acceleration time (s) = 1 unit is 100ms
Byte6: Deceleration time (s) =  1 unit is 100ms

CAN ID X value for the different Node ID:
41 - 9		42 - A 		43-B
	
	***UPDATES***
V2:
1. RPM transmit delay has been added after Ignition turns on..
2. CAN_TX block has been changerd to CAN_TX_ENH.
3. Temporary Phase current limit has been added to var input
V3
1. Added Ignition state bit as VAR_OUTPUT.
V4
1. UPDATED AVG RPM TO 75 TO HOLD ON THE MCU.
2. RPM DELAY TIME REDUCED TO 250MS
*)
VAR_INPUT
	CAN_CHANNEL: BYTE;
	ID_22X: DWORD;
	TARGET_RPM: INT;
	REFERNCE_RPM: INT;
	RAMP: INT;
	MCU_RAMP: BYTE;
	HILL_HOLD_IN: BOOL;
	PHASE_CURRENT_LIMIT: BYTE;
END_VAR
VAR
	IGNITION_ON: BOOL;
	IGNITION_STATE: BYTE;
	HOLD_ON: BOOL;
	ABS_RPM: INT;
	RPM_RAMP: RAMP_INT;
	WB_TARGET_RPM: WORD_BYTE_CONVERSION;
	PACK_TX: PACK_BYTES;
	TX: CAN_TX_ENH;
	RPM_DELAY: TON;
	TIMER: TON;
END_VAR
VAR_OUTPUT
	TARGET_RPM_OUT: INT;
	IGNITION_OUT: BOOL;
END_VAR
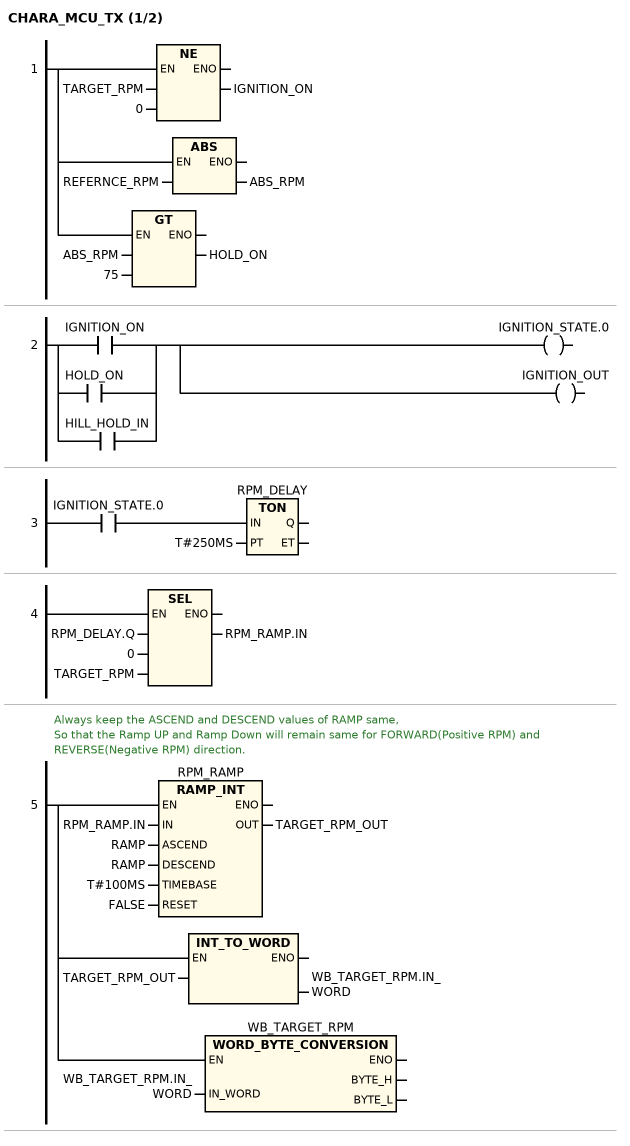
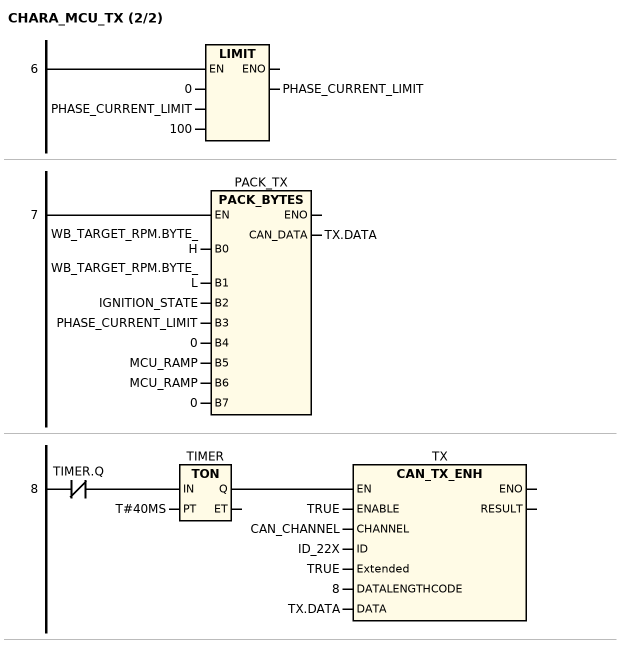
_LD_ (* Ladder Diagram *)
NETWORK 1
	*
		EN --- NE(TARGET_RPM, 0) => IGNITION_ON
		EN --- ABS(REFERNCE_RPM) => ABS_RPM
		EN --- GT(ABS_RPM, 75) => HOLD_ON
NETWORK 2
	{ [IGNITION_ON] | [HOLD_ON] | [HILL_HOLD_IN] } --- (IGNITION_STATE.0) (IGNITION_OUT)
NETWORK 3
	[IGNITION_STATE.0] - RPM_DELAY:TON(IN: *, PT: T#250MS)
NETWORK 4
	*
		EN --- SEL(RPM_DELAY.Q, 0, TARGET_RPM) => RPM_RAMP.IN
NETWORK 5 (* Always keep the ASCEND and DESCEND values of RAMP same, / So that the Ramp UP and Ramp Down will remain same for FORWARD(Positive RPM) and REVERSE(Negative RPM) direction. *)
	*
		EN --- RPM_RAMP:RAMP_INT(IN: RPM_RAMP.IN, ASCEND: RAMP, DESCEND: RAMP, TIMEBASE: T#100MS, RESET: FALSE) => TARGET_RPM_OUT
		EN --- INT_TO_WORD(TARGET_RPM_OUT) => WB_TARGET_RPM.IN_WORD
		EN --- WB_TARGET_RPM:WORD_BYTE_CONVERSION(IN_WORD: WB_TARGET_RPM.IN_WORD)
NETWORK 6
	*
		EN --- LIMIT(0, PHASE_CURRENT_LIMIT, 100) => PHASE_CURRENT_LIMIT
NETWORK 7
	*
		EN --- PACK_TX:PACK_BYTES(B0: WB_TARGET_RPM.BYTE_H, B1: WB_TARGET_RPM.BYTE_L, B2: IGNITION_STATE, B3: PHASE_CURRENT_LIMIT, B4: 0, B5: MCU_RAMP, B6: MCU_RAMP, B7: 0) => TX.DATA
NETWORK 8
	[/TIMER.Q] - TIMER:TON(IN: *, PT: T#40MS)
		EN --- TX:CAN_TX_ENH(ENABLE: TRUE, CHANNEL: CAN_CHANNEL, ID: ID_22X, Extended: TRUE, DATALENGTHCODE: 8, DATA: TX.DATA)
_END_LD_
(* the same logic as Structured Text *)
(* Network 1 *)
IGNITION_ON := TARGET_RPM <> 0;
ABS_RPM := ABS(REFERNCE_RPM);
HOLD_ON := ABS_RPM > 75;
(* Network 2 *)
IGNITION_STATE.0 := IGNITION_ON OR HOLD_ON OR HILL_HOLD_IN;
IGNITION_OUT := IGNITION_STATE.0;
(* Network 3 *)
RPM_DELAY(IN := IGNITION_STATE.0, PT := T#250MS);
(* Network 4 *)
RPM_RAMP.IN := SEL(RPM_DELAY.Q, 0, TARGET_RPM);
(* Network 5: Always keep the ASCEND and DESCEND values of RAMP same, / So that the Ramp UP and Ramp Down will remain same for FORWARD(Positive RPM) and REVERSE(Negative RPM) direction. *)
RPM_RAMP(IN := RPM_RAMP.IN, ASCEND := RAMP, DESCEND := RAMP, TIMEBASE := T#100MS, RESET := FALSE);
TARGET_RPM_OUT := RPM_RAMP.OUT;
WB_TARGET_RPM.IN_WORD := INT_TO_WORD(TARGET_RPM_OUT);
WB_TARGET_RPM(IN_WORD := WB_TARGET_RPM.IN_WORD);
(* Network 6 *)
PHASE_CURRENT_LIMIT := LIMIT(0, PHASE_CURRENT_LIMIT, 100);
(* Network 7 *)
PACK_TX(B0 := WB_TARGET_RPM.BYTE_H, B1 := WB_TARGET_RPM.BYTE_L, B2 := IGNITION_STATE, B3 := PHASE_CURRENT_LIMIT, B4 := 0, B5 := MCU_RAMP, B6 := MCU_RAMP, B7 := 0);
TX.DATA := PACK_TX.CAN_DATA;
(* Network 8 *)
TIMER(IN := NOT TIMER.Q, PT := T#40MS);
IF TIMER.Q THEN
	TX(ENABLE := TRUE, CHANNEL := CAN_CHANNEL, ID := ID_22X, Extended := TRUE, DATALENGTHCODE := 8, DATA := TX.DATA);
END_IF;
END_FUNCTION_BLOCK

(* POU FB_LIBRARY/WORD_BYTE_CONVERSION, FBD *)
FUNCTION_BLOCK WORD_BYTE_CONVERSION
(*
Created by: Bhagyesh Unadkat
Date: 29-03-24
Version: 1
Updated by:
Update date:
Description: This block converts the WORD data into two BYTEs
*)
VAR_INPUT
	IN_WORD: WORD;
END_VAR
VAR_OUTPUT
	BYTE_H: BYTE;
	BYTE_L: BYTE;
END_VAR
VAR
END_VAR
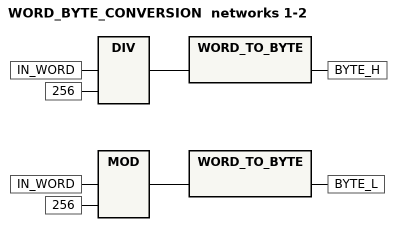
_FBD_ (* Function Block Diagram *)
NETWORK 1
	WORD_TO_BYTE(DIV(IN_WORD, 256)) => BYTE_H
NETWORK 2
	WORD_TO_BYTE(MOD(IN_WORD, 256)) => BYTE_L
_END_FBD_
(* the same logic as Structured Text *)
(* Network 1 *)
BYTE_H := WORD_TO_BYTE(IN_WORD / 256);
(* Network 2 *)
BYTE_L := WORD_TO_BYTE(IN_WORD MOD 256);
END_FUNCTION_BLOCK

(* POU FB_LIBRARY/PACK_BYTES, ST *)
FUNCTION_BLOCK PACK_BYTES
(*
Created by: Bhagyesh Unadkat
Date: 29-03-24
Version: 1
Updated by:
Update date:
Description: This block merges 8 bytes of data into 1 CAN data array.
*)
VAR_INPUT
	B0: BYTE;
	B1: BYTE;
	B2: BYTE;
	B3: BYTE;
	B4: BYTE;
	B5: BYTE;
	B6: BYTE;
	B7: BYTE;
END_VAR
VAR_OUTPUT
	CAN_DATA: ARRAY [0..7] OF BYTE;
END_VAR
CAN_DATA[0]:= B0;
CAN_DATA[1]:= B1;
CAN_DATA[2]:= B2;
CAN_DATA[3]:= B3;
CAN_DATA[4]:= B4;
CAN_DATA[5]:= B5;
CAN_DATA[6]:= B6;
CAN_DATA[7]:= B7;
END_FUNCTION_BLOCK

(* POU PROGRAM_FBs/CLN_BATTERY, LD *)
FUNCTION_BLOCK CLN_BATTERY
(*
Created by: Anirudh Raghavan
Date: 10-01-24
Version: 4
Updated by: Bhagyesh
Update date: 15-09-2024
Description: This block reads the data of CLN Battery.
	
	*** UPDATES ***
V3: 
	Removed the SOC mapping function.
V4
	Variable modifiacations and faults removed
*)
VAR_INPUT
	CAN_CHANNEL: BYTE;
END_VAR
VAR_OUTPUT
	SOC: BYTE;
	SOH: BYTE;
       CURRENT: INT;
	CHARGING: BOOL;
	POWER: INT; (*Watt*)
	NTC_1: BYTE;
	NTC_2: BYTE;
	TOTAL_CAPACITY: INT; (*Ah*)
	CAPACITY: INT; (*Ah*)
	CAN_ERROR: BOOL;

END_VAR
VAR
	RX_205: RX_CAN;
	RX_1E1: RX_CAN;
	RX_1F5: RX_CAN;
	RX_357: RX_CAN;
	DELAY: TON;
	SOC_WORD: WORD;
	SOH_WORD: WORD;
	VOLTAGE_WORD: WORD;
	CURRENT_WORD: WORD;
	VOLTAGE: INT;
	CAPACITY_WORD: WORD;
	CAPACITY_AH: WORD;
	TOTAL_CAPACITY_WORD: WORD;
	TOTAL_CAPACITY_AH: WORD;

END_VAR
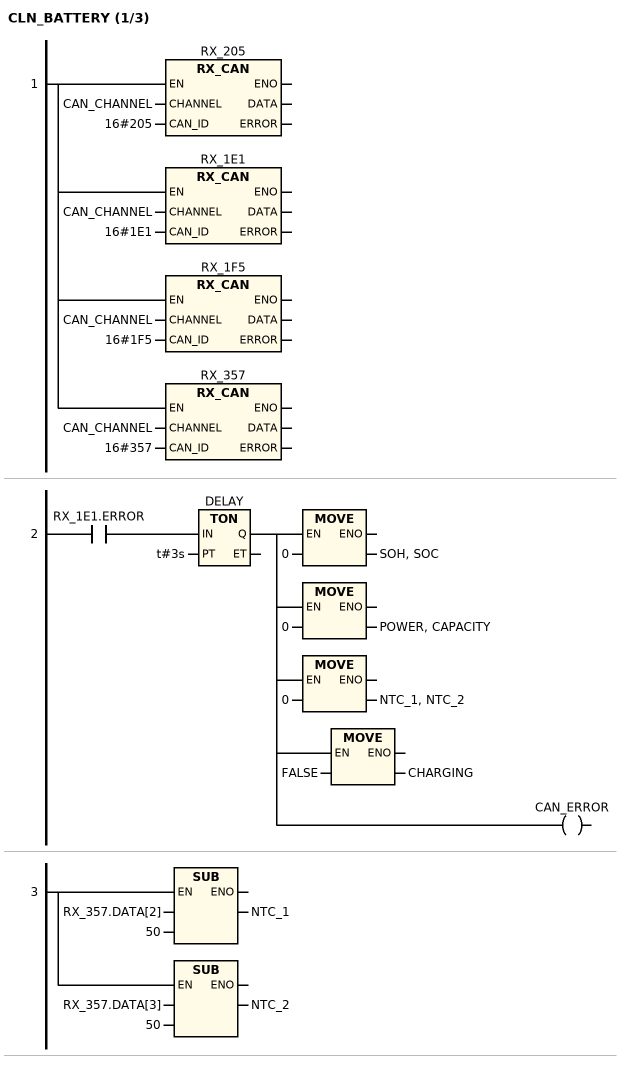
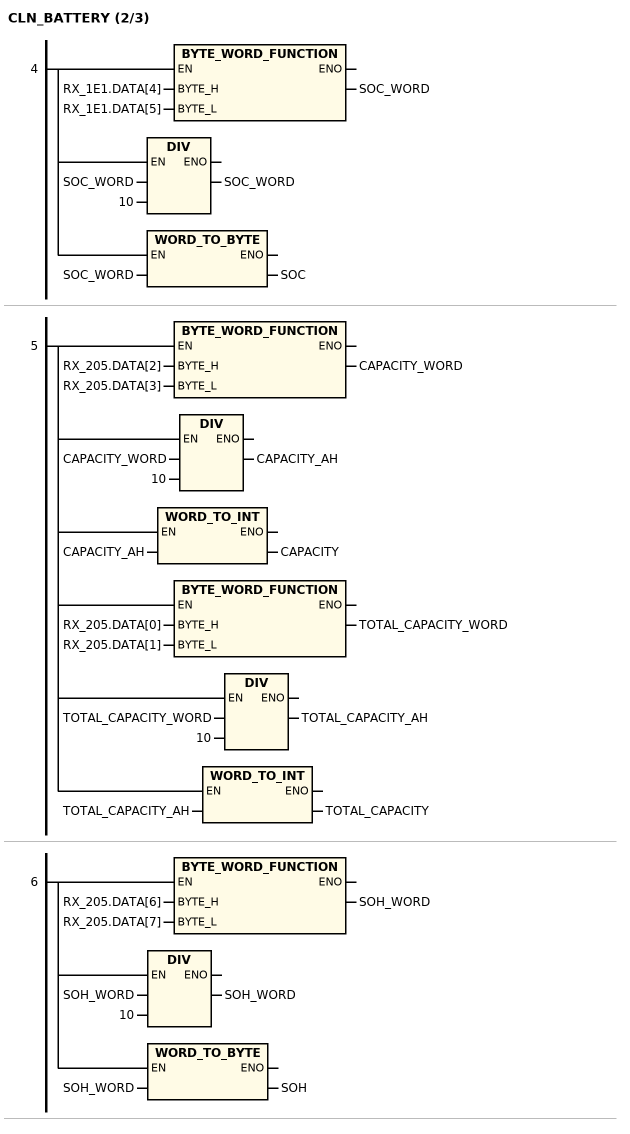
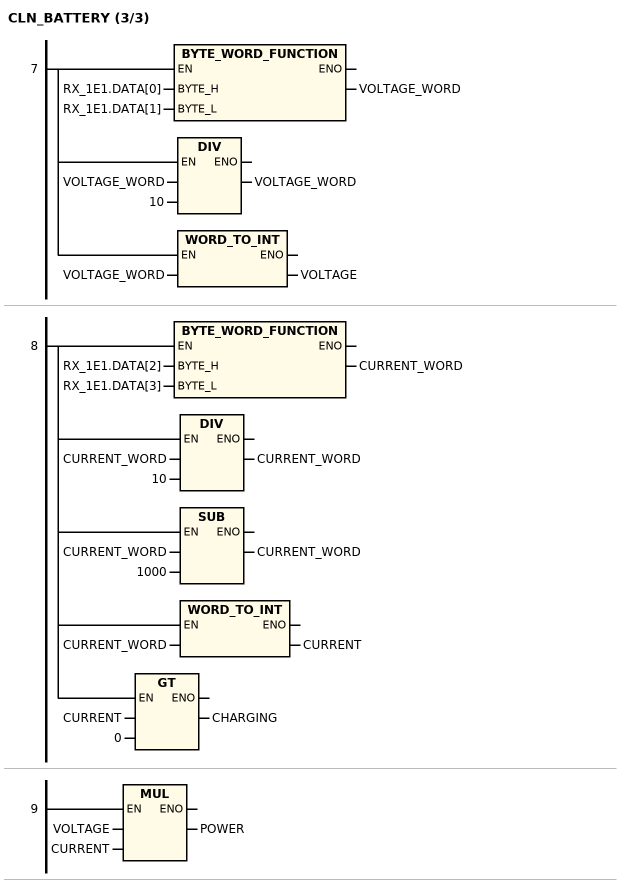
_LD_ (* Ladder Diagram *)
NETWORK 1
	*
		EN --- RX_205:RX_CAN(CHANNEL: CAN_CHANNEL, CAN_ID: 16#205)
		EN --- RX_1E1:RX_CAN(CHANNEL: CAN_CHANNEL, CAN_ID: 16#1E1)
		EN --- RX_1F5:RX_CAN(CHANNEL: CAN_CHANNEL, CAN_ID: 16#1F5)
		EN --- RX_357:RX_CAN(CHANNEL: CAN_CHANNEL, CAN_ID: 16#357)
NETWORK 2
	[RX_1E1.ERROR] - DELAY:TON(IN: *, PT: t#3s) --- (CAN_ERROR)
		EN --- MOVE(0) => SOH, SOC
		EN --- MOVE(0) => POWER, CAPACITY
		EN --- MOVE(0) => NTC_1, NTC_2
		EN --- MOVE(FALSE) => CHARGING
NETWORK 3
	*
		EN --- SUB(RX_357.DATA[2], 50) => NTC_1
		EN --- SUB(RX_357.DATA[3], 50) => NTC_2
NETWORK 4
	*
		EN --- BYTE_WORD_FUNCTION(BYTE_H: RX_1E1.DATA[4], BYTE_L: RX_1E1.DATA[5]) => SOC_WORD
		EN --- DIV(SOC_WORD, 10) => SOC_WORD
		EN --- WORD_TO_BYTE(SOC_WORD) => SOC
NETWORK 5
	*
		EN --- BYTE_WORD_FUNCTION(BYTE_H: RX_205.DATA[2], BYTE_L: RX_205.DATA[3]) => CAPACITY_WORD
		EN --- DIV(CAPACITY_WORD, 10) => CAPACITY_AH
		EN --- WORD_TO_INT(CAPACITY_AH) => CAPACITY
		EN --- BYTE_WORD_FUNCTION(BYTE_H: RX_205.DATA[0], BYTE_L: RX_205.DATA[1]) => TOTAL_CAPACITY_WORD
		EN --- DIV(TOTAL_CAPACITY_WORD, 10) => TOTAL_CAPACITY_AH
		EN --- WORD_TO_INT(TOTAL_CAPACITY_AH) => TOTAL_CAPACITY
NETWORK 6
	*
		EN --- BYTE_WORD_FUNCTION(BYTE_H: RX_205.DATA[6], BYTE_L: RX_205.DATA[7]) => SOH_WORD
		EN --- DIV(SOH_WORD, 10) => SOH_WORD
		EN --- WORD_TO_BYTE(SOH_WORD) => SOH
NETWORK 7
	*
		EN --- BYTE_WORD_FUNCTION(BYTE_H: RX_1E1.DATA[0], BYTE_L: RX_1E1.DATA[1]) => VOLTAGE_WORD
		EN --- DIV(VOLTAGE_WORD, 10) => VOLTAGE_WORD
		EN --- WORD_TO_INT(VOLTAGE_WORD) => VOLTAGE
NETWORK 8
	*
		EN --- BYTE_WORD_FUNCTION(BYTE_H: RX_1E1.DATA[2], BYTE_L: RX_1E1.DATA[3]) => CURRENT_WORD
		EN --- DIV(CURRENT_WORD, 10) => CURRENT_WORD
		EN --- SUB(CURRENT_WORD, 1000) => CURRENT_WORD
		EN --- WORD_TO_INT(CURRENT_WORD) => CURRENT
		EN --- GT(CURRENT, 0) => CHARGING
NETWORK 9
	*
		EN --- MUL(VOLTAGE, CURRENT) => POWER
_END_LD_
(* the same logic as Structured Text *)
(* Network 1 *)
RX_205(CHANNEL := CAN_CHANNEL, CAN_ID := 16#205);
RX_1E1(CHANNEL := CAN_CHANNEL, CAN_ID := 16#1E1);
RX_1F5(CHANNEL := CAN_CHANNEL, CAN_ID := 16#1F5);
RX_357(CHANNEL := CAN_CHANNEL, CAN_ID := 16#357);
(* Network 2: see the listing above *)
(* Network 3 *)
NTC_1 := RX_357.DATA[2] - 50;
NTC_2 := RX_357.DATA[3] - 50;
(* Network 4 *)
SOC_WORD := BYTE_WORD_FUNCTION(BYTE_H := RX_1E1.DATA[4], BYTE_L := RX_1E1.DATA[5]);
SOC_WORD := SOC_WORD / 10;
SOC := WORD_TO_BYTE(SOC_WORD);
(* Network 5 *)
CAPACITY_WORD := BYTE_WORD_FUNCTION(BYTE_H := RX_205.DATA[2], BYTE_L := RX_205.DATA[3]);
CAPACITY_AH := CAPACITY_WORD / 10;
CAPACITY := WORD_TO_INT(CAPACITY_AH);
TOTAL_CAPACITY_WORD := BYTE_WORD_FUNCTION(BYTE_H := RX_205.DATA[0], BYTE_L := RX_205.DATA[1]);
TOTAL_CAPACITY_AH := TOTAL_CAPACITY_WORD / 10;
TOTAL_CAPACITY := WORD_TO_INT(TOTAL_CAPACITY_AH);
(* Network 6 *)
SOH_WORD := BYTE_WORD_FUNCTION(BYTE_H := RX_205.DATA[6], BYTE_L := RX_205.DATA[7]);
SOH_WORD := SOH_WORD / 10;
SOH := WORD_TO_BYTE(SOH_WORD);
(* Network 7 *)
VOLTAGE_WORD := BYTE_WORD_FUNCTION(BYTE_H := RX_1E1.DATA[0], BYTE_L := RX_1E1.DATA[1]);
VOLTAGE_WORD := VOLTAGE_WORD / 10;
VOLTAGE := WORD_TO_INT(VOLTAGE_WORD);
(* Network 8 *)
CURRENT_WORD := BYTE_WORD_FUNCTION(BYTE_H := RX_1E1.DATA[2], BYTE_L := RX_1E1.DATA[3]);
CURRENT_WORD := CURRENT_WORD / 10;
CURRENT_WORD := CURRENT_WORD - 1000;
CURRENT := WORD_TO_INT(CURRENT_WORD);
CHARGING := CURRENT > 0;
(* Network 9 *)
POWER := VOLTAGE * CURRENT;
END_FUNCTION_BLOCK

(* POU PROGRAM_FBs/CLN_BATTERY_SELECTION, LD *)
FUNCTION_BLOCK CLN_BATTERY_SELECTION
(*
Created BY: Adiga
Date: 25-01-24
Version: 1
      
*)

VAR_INPUT
	BAT_SOC: BYTE;
	BAT_SOH: BYTE;
	BAT_POWER: INT;
	BAT_NTC1: BYTE;
	BAT_NTC2: BYTE;
	BAT_CAN_ERROR: BOOL;
	BATTERY_CAPACITY_WORD: WORD;
	BAT_CURRENT: INT;
END_VAR
VAR_OUTPUT
	LOW_SOC: BOOL;
END_VAR
VAR
	RTRIG_B1: R_TRIG;
	RTRIG_B2: R_TRIG;
	BAT_1: BOOL;
	BAT_2: BOOL;
	SOC_INT: INT;
	SOC_MAP: INT;
	SOC: BYTE;

	TON1: TON;
	TON2: TON;
END_VAR
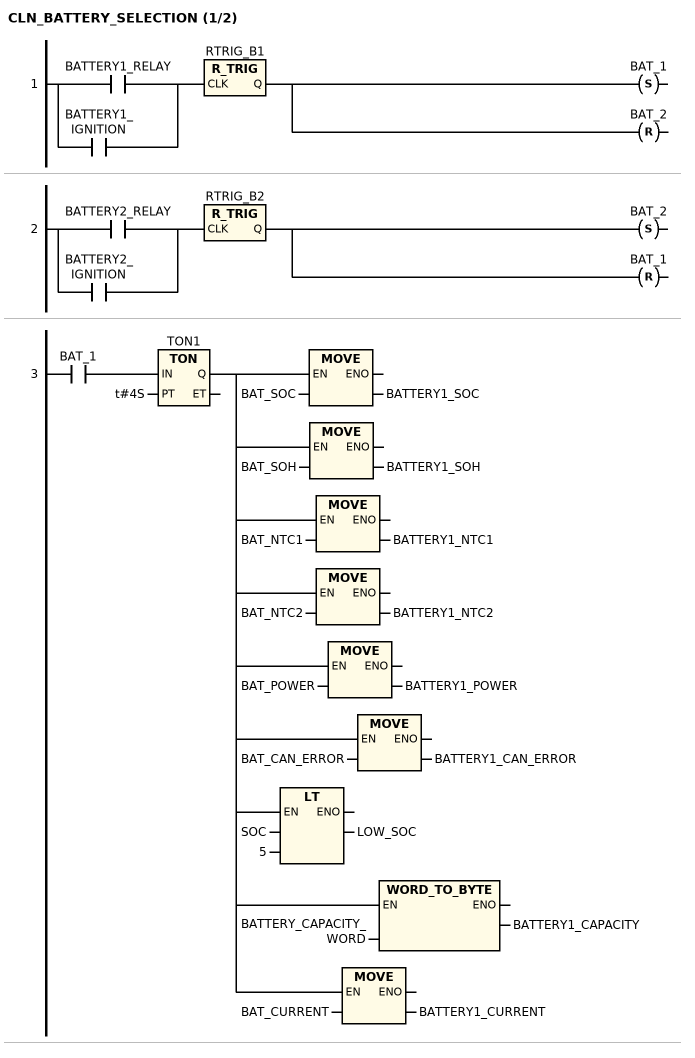
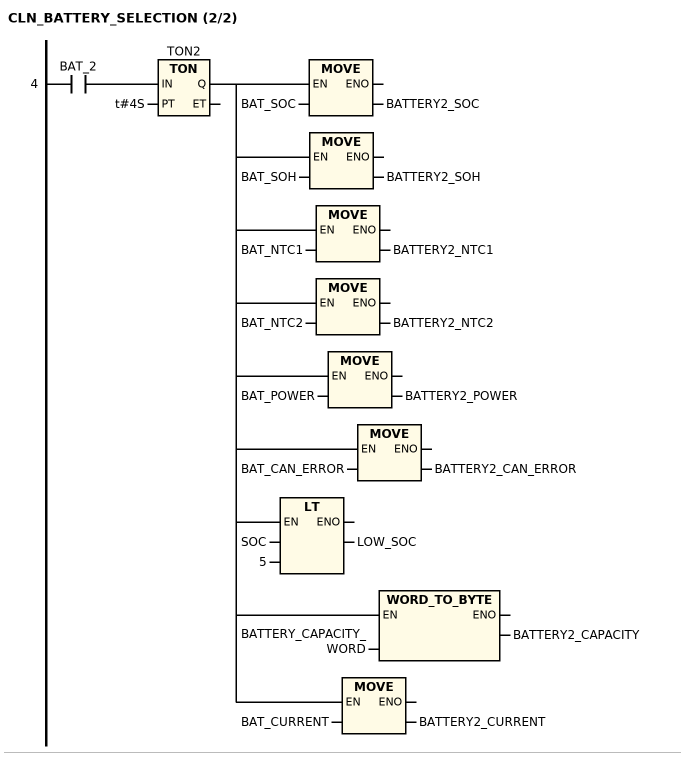
_LD_ (* Ladder Diagram *)
NETWORK 1
	{ [BATTERY1_RELAY] | [BATTERY1_IGNITION] } - RTRIG_B1:R_TRIG(CLK: *) --- (S BAT_1) (R BAT_2)
NETWORK 2
	{ [BATTERY2_RELAY] | [BATTERY2_IGNITION] } - RTRIG_B2:R_TRIG(CLK: *) --- (S BAT_2) (R BAT_1)
NETWORK 3
	[BAT_1] - TON1:TON(IN: *, PT: t#4S)
		EN --- MOVE(BAT_SOC) => BATTERY1_SOC
		EN --- MOVE(BAT_SOH) => BATTERY1_SOH
		EN --- MOVE(BAT_NTC1) => BATTERY1_NTC1
		EN --- MOVE(BAT_NTC2) => BATTERY1_NTC2
		EN --- MOVE(BAT_POWER) => BATTERY1_POWER
		EN --- MOVE(BAT_CAN_ERROR) => BATTERY1_CAN_ERROR
		EN --- LT(SOC, 5) => LOW_SOC
		EN --- WORD_TO_BYTE(BATTERY_CAPACITY_WORD) => BATTERY1_CAPACITY
		EN --- MOVE(BAT_CURRENT) => BATTERY1_CURRENT
NETWORK 4
	[BAT_2] - TON2:TON(IN: *, PT: t#4S)
		EN --- MOVE(BAT_SOC) => BATTERY2_SOC
		EN --- MOVE(BAT_SOH) => BATTERY2_SOH
		EN --- MOVE(BAT_NTC1) => BATTERY2_NTC1
		EN --- MOVE(BAT_NTC2) => BATTERY2_NTC2
		EN --- MOVE(BAT_POWER) => BATTERY2_POWER
		EN --- MOVE(BAT_CAN_ERROR) => BATTERY2_CAN_ERROR
		EN --- LT(SOC, 5) => LOW_SOC
		EN --- WORD_TO_BYTE(BATTERY_CAPACITY_WORD) => BATTERY2_CAPACITY
		EN --- MOVE(BAT_CURRENT) => BATTERY2_CURRENT
_END_LD_
(* the same logic as Structured Text *)
(* Network 1 *)
RTRIG_B1(CLK := BATTERY1_RELAY OR BATTERY1_IGNITION);
IF RTRIG_B1.Q THEN BAT_1 := TRUE; BAT_2 := FALSE; END_IF;
(* Network 2 *)
RTRIG_B2(CLK := BATTERY2_RELAY OR BATTERY2_IGNITION);
IF RTRIG_B2.Q THEN BAT_2 := TRUE; BAT_1 := FALSE; END_IF;
(* Network 3 *)
TON1(IN := BAT_1, PT := t#4S);
IF TON1.Q THEN
	BATTERY1_SOC := BAT_SOC;
	BATTERY1_SOH := BAT_SOH;
	BATTERY1_NTC1 := BAT_NTC1;
	BATTERY1_NTC2 := BAT_NTC2;
	BATTERY1_POWER := BAT_POWER;
	BATTERY1_CAN_ERROR := BAT_CAN_ERROR;
	LOW_SOC := SOC < 5;
	BATTERY1_CAPACITY := WORD_TO_BYTE(BATTERY_CAPACITY_WORD);
	BATTERY1_CURRENT := BAT_CURRENT;
END_IF;
(* Network 4 *)
TON2(IN := BAT_2, PT := t#4S);
IF TON2.Q THEN
	BATTERY2_SOC := BAT_SOC;
	BATTERY2_SOH := BAT_SOH;
	BATTERY2_NTC1 := BAT_NTC1;
	BATTERY2_NTC2 := BAT_NTC2;
	BATTERY2_POWER := BAT_POWER;
	BATTERY2_CAN_ERROR := BAT_CAN_ERROR;
	LOW_SOC := SOC < 5;
	BATTERY2_CAPACITY := WORD_TO_BYTE(BATTERY_CAPACITY_WORD);
	BATTERY2_CURRENT := BAT_CURRENT;
END_IF;
END_FUNCTION_BLOCK

(* POU PROGRAM_FBs/CLN_BATTERY_SELECTION_2, LD *)
 FUNCTION_BLOCK CLN_BATTERY_SELECTION_2
VAR_INPUT
	BAT_SOC: BYTE;
	BAT_SOH: BYTE;
	BAT_POWER: INT;
	BAT_NTC1: BYTE;
	BAT_NTC2: BYTE;
	BAT_CAN_ERROR: BOOL;
	BAT_CURRENT: INT;
END_VAR
VAR_OUTPUT
END_VAR
VAR
	BAT1_TON: TON;
	BAT2_TON: TON;
END_VAR
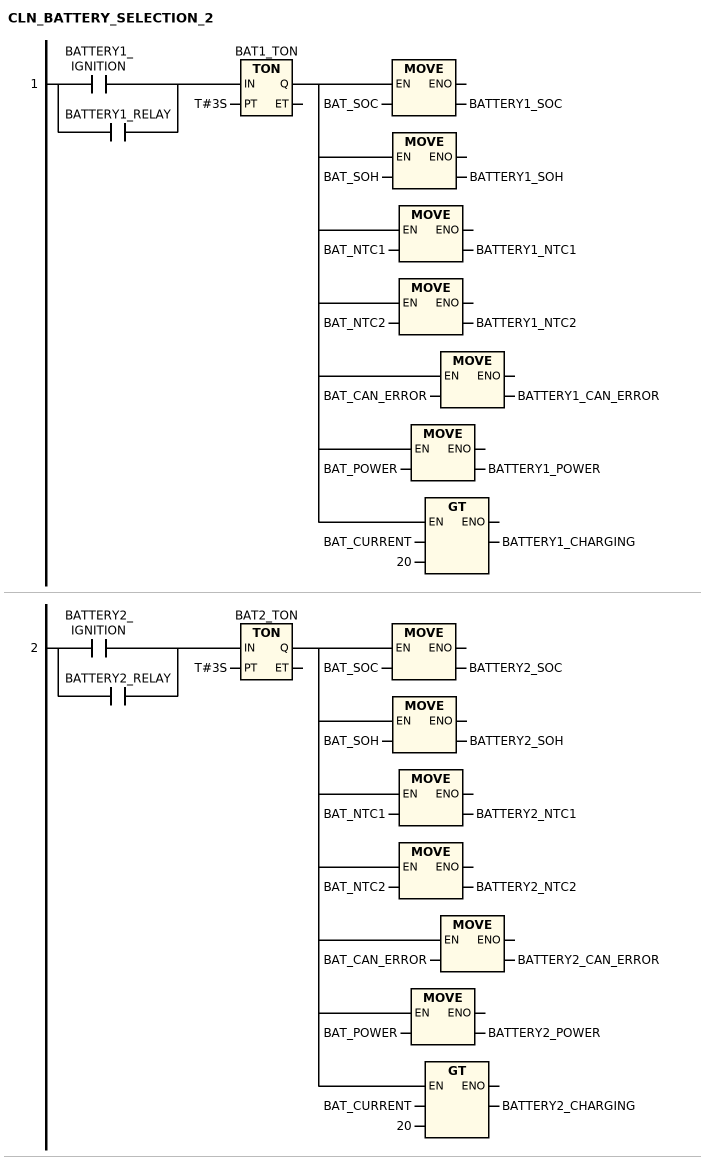
_LD_ (* Ladder Diagram *)
NETWORK 1
	{ [BATTERY1_IGNITION] | [BATTERY1_RELAY] } - BAT1_TON:TON(IN: *, PT: T#3S)
		EN --- MOVE(BAT_SOC) => BATTERY1_SOC
		EN --- MOVE(BAT_SOH) => BATTERY1_SOH
		EN --- MOVE(BAT_NTC1) => BATTERY1_NTC1
		EN --- MOVE(BAT_NTC2) => BATTERY1_NTC2
		EN --- MOVE(BAT_CAN_ERROR) => BATTERY1_CAN_ERROR
		EN --- MOVE(BAT_POWER) => BATTERY1_POWER
		EN --- GT(BAT_CURRENT, 20) => BATTERY1_CHARGING
NETWORK 2
	{ [BATTERY2_IGNITION] | [BATTERY2_RELAY] } - BAT2_TON:TON(IN: *, PT: T#3S)
		EN --- MOVE(BAT_SOC) => BATTERY2_SOC
		EN --- MOVE(BAT_SOH) => BATTERY2_SOH
		EN --- MOVE(BAT_NTC1) => BATTERY2_NTC1
		EN --- MOVE(BAT_NTC2) => BATTERY2_NTC2
		EN --- MOVE(BAT_CAN_ERROR) => BATTERY2_CAN_ERROR
		EN --- MOVE(BAT_POWER) => BATTERY2_POWER
		EN --- GT(BAT_CURRENT, 20) => BATTERY2_CHARGING
_END_LD_
(* the same logic as Structured Text *)
(* Network 1 *)
BAT1_TON(IN := BATTERY1_IGNITION OR BATTERY1_RELAY, PT := T#3S);
IF BAT1_TON.Q THEN
	BATTERY1_SOC := BAT_SOC;
	BATTERY1_SOH := BAT_SOH;
	BATTERY1_NTC1 := BAT_NTC1;
	BATTERY1_NTC2 := BAT_NTC2;
	BATTERY1_CAN_ERROR := BAT_CAN_ERROR;
	BATTERY1_POWER := BAT_POWER;
	BATTERY1_CHARGING := BAT_CURRENT > 20;
END_IF;
(* Network 2 *)
BAT2_TON(IN := BATTERY2_IGNITION OR BATTERY2_RELAY, PT := T#3S);
IF BAT2_TON.Q THEN
	BATTERY2_SOC := BAT_SOC;
	BATTERY2_SOH := BAT_SOH;
	BATTERY2_NTC1 := BAT_NTC1;
	BATTERY2_NTC2 := BAT_NTC2;
	BATTERY2_CAN_ERROR := BAT_CAN_ERROR;
	BATTERY2_POWER := BAT_POWER;
	BATTERY2_CHARGING := BAT_CURRENT > 20;
END_IF;
END_FUNCTION_BLOCK

(* POU PROGRAM_FBs/CLN_BATTERY_SWITCH, LD *)
FUNCTION_BLOCK CLN_BATTERY_SWITCH

(*THIS BLOCK IS COMPATIBLE FOR 2X CLN BATTERIES*)

VAR_INPUT
	CHARGER_IN: BOOL;
	IGN_KEY: BOOL;
	BAT1_IGNITION: BOOL;
	BAT2_IGNITION: BOOL;
	SOC_BAT1: BYTE;
	SOC_BAT2: BYTE;
	BAT1_CAN_ERROR: BOOL;
	BAT2_CAN_ERROR: BOOL;
END_VAR

VAR_OUTPUT
	RELAY_BAT1: BOOL;
	RELAY_BAT2: BOOL;
	ERROR: BOOL;
END_VAR

VAR
	BAT1_CAN_TIMER: TON;
	BAT2_CAN_TIMER: TON;
	BAT1_FULL: BOOL;
	BAT2_FULL: BOOL;
	BAT1_80: BOOL;
	BAT2_80: BOOL;
	CHARGE_1: BOOL;
	RELAY1_TIMER: TON;
	RELAY2_TIMER: TON;
	BLUE_BLINK: BLINK;
	CHARGE1_BLINK: BLINK;
	CHARGE2_BLINK: BLINK;
	CHARGING_SAFETY: BOOL;

	ERROR_TIMER: TON;
END_VAR
